KUKA KRL program: EPS_2_251806_MH46A_A_20260213065142.src

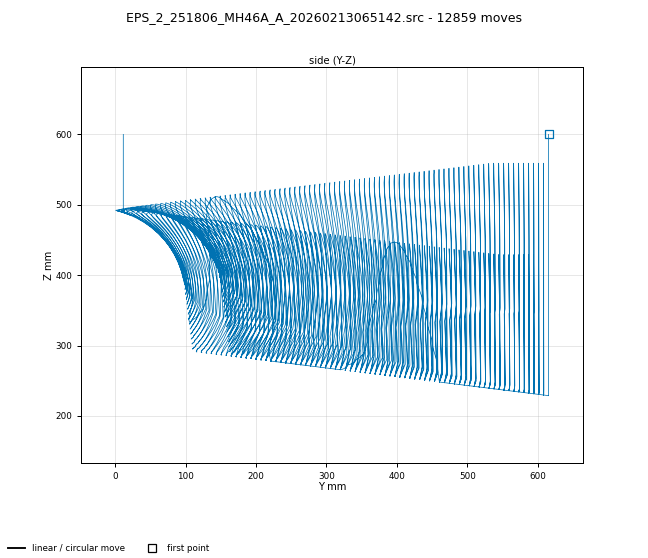
[picture p0: tool path of EPS_2_251806_MH46A_A_20260213065142.src, 12859 of 12861 moves have a stored position in this frame; points joined in program order, loops and branches not executed]
&ACCESS RVP
&REL 4
&COMMENT QRS 19112012
&PARAM EDITMASK = *
DEF PART()
EXT BAS (BAS_COMMAND :IN,REAL :IN )
INT I
BAS (#INITMOV,0 )

;KUKA QRS Post kuka4.cps  Date:22-06-2017 !

File_ID=3033

QRS_PRE_INIT()

;Init var - Until changes are made in qrs_pre_init
Outlet_Square_prg=0
Inlet_1_Square_prg=0
Inlet_2_Square_prg=0
Inlet_3_Square_prg=0
Inlet_4_Square_prg=0
Inlet_5_Square_prg=0

Outlet_1={X 0.000, Y 535.490, Z 458.500, B 0.000, E1 0.000 }
Inlet_1={X 0.000, Y 544.760, Z 328.500, B 0.000, E1 188.000 }
Outlet_1_type=201
Inlet_1_type=201
;QRS#1=Sidecore dimensions
;QRS#2=200-8" PVC SDR 35
;QRS#3=200-8" PVC SDR 35
;QRS#4=
;QRS#5=
;QRS#6=
;QRS#7=
;QRS#8=
;QRS#9=12-08 PSX
;QRS#10=12-08 PSX
;QRS#11=
;QRS#12=
;QRS#13=
;QRS#14=
;QRS#15=
;QRS#16=1220x127x838 2,75'
;QRS#17=EPS Height
;QRS#18=559
;QRS#19=*
;QRS#20= UPDATED VERSION 22-06-2017
;QRS#21=*
Outlet_Square=0100
Inlet_1_Square=0100
Inlet_2_Square=0
Inlet_3_Square=0
Inlet_4_Square=0
Inlet_5_Square=0
Mill_Square=1
Outlet_Square_Prg=204
Inlet_1_Square_prg=204

QRS_INIT()

$ADVANCE=5

; T1
PTP {E1 173.608,E2 173.608}
PTP {X 0,Y 615.502,A -85,B 0,C 180,E1 173.608,E2 173.608,E3 0,E4 0,E5 0,E6 0}
QRS_SPEED_INIT()
LIN {X 0,Y 615.502,Z 600,A -85,B 0,C 180,E1 173.608,E2 173.608,E3 0,E4 0,E5 0,E6 0} C_VEL
LIN {X 0,Y 615.502,Z 238.877,A -85,B 0,C 180,E1 173.608,E2 173.608} C_VEL
LIN {X 0,Y 615.502,Z 230.7,A -85,B 0,C 180,E1 173.608,E2 173.608} C_VEL
LIN {X 0,Y 615.471,Z 228.7,A -85,B 0,C 180,E1 173.422,E2 173.422} C_VEL
LIN {X 0,Y 615.413,Z 228.7,A -85,B 0,C 180,E1 170.8,E2 170.8} C_VEL
LIN {X 0,Y 615.412,Z 228.7,A -85,B 0,C 180,E1 168.805,E2 168.805} C_VEL
LIN {X 0,Y 615.411,Z 228.7,A -85,B 0,C 180,E1 166.797,E2 166.797} C_VEL
LIN {X 0,Y 615.451,Z 228.7,A -85,B 0,C 180,E1 164.094,E2 164.094} C_VEL
LIN {X 0,Y 615.438,Z 228.7,A -85,B 0,C 180,E1 161.352,E2 161.352} C_VEL
LIN {X 0,Y 615.424,Z 228.701,A -85,B 0,C 180,E1 159.267,E2 159.267} C_VEL
LIN {X 0,Y 615.418,Z 228.7,A -85,B 0,C 180,E1 157.152,E2 157.152} C_VEL
LIN {X 0,Y 615.412,Z 228.7,A -85,B 0,C 180,E1 155.005,E2 155.005} C_VEL
LIN {X 0,Y 615.413,Z 228.7,A -85,B 0,C 180,E1 152.819,E2 152.819} C_VEL
LIN {X 0,Y 615.467,Z 228.7,A -85,B 0,C 180,E1 150.206,E2 150.206} C_VEL
LIN {X 0,Y 615.434,Z 228.7,A -85,B 0,C 180,E1 147.539,E2 147.539} C_VEL
LIN {X 0,Y 615.411,Z 228.7,A -85,B 0,C 180,E1 145.18,E2 145.18} C_VEL
LIN {X 0,Y 615.411,Z 228.7,A -85,B 0,C 180,E1 143.071,E2 143.071} C_VEL
LIN {X 0,Y 615.415,Z 228.7,A -85,B 0,C 180,E1 140.944,E2 140.944} C_VEL
LIN {X 0,Y 615.451,Z 228.7,A -85,B 0,C 180,E1 138.523,E2 138.523} C_VEL
LIN {X 0,Y 615.443,Z 228.701,A -85,B 0,C 180,E1 135.846,E2 135.846} C_VEL
LIN {X 0,Y 615.461,Z 228.7,A -85,B 0,C 180,E1 133.994,E2 133.994} C_VEL
LIN {X 0,Y 615.414,Z 228.7,A -85,B 0,C 180,E1 131.478,E2 131.478} C_VEL
LIN {X 0,Y 615.429,Z 228.7,A -85,B 0,C 180,E1 128.907,E2 128.907} C_VEL
LIN {X 0,Y 615.472,Z 228.705,A -85,B 0,C 180,E1 126.425,E2 126.425} C_VEL
LIN {X 0,Y 615.44,Z 228.701,A -85,B 0,C 180,E1 124.024,E2 124.024} C_VEL
LIN {X 0,Y 615.416,Z 228.7,A -85,B 0,C 180,E1 121.688,E2 121.688} C_VEL
LIN {X 0,Y 615.412,Z 228.7,A -85,B 0,C 180,E1 119.409,E2 119.409} C_VEL
LIN {X 0,Y 615.435,Z 228.699,A -85,B 0,C 180,E1 117.034,E2 117.034} C_VEL
LIN {X 0,Y 615.454,Z 228.7,A -85,B 0,C 180,E1 114.273,E2 114.273} C_VEL
LIN {X 0,Y 615.436,Z 228.7,A -85,B 0,C 180,E1 112.138,E2 112.138} C_VEL
LIN {X 0,Y 615.425,Z 228.7,A -85,B 0,C 180,E1 110.034,E2 110.034} C_VEL
LIN {X 0,Y 615.418,Z 228.7,A -85,B 0,C 180,E1 107.958,E2 107.958} C_VEL
LIN {X 0,Y 615.415,Z 228.7,A -85,B 0,C 180,E1 105.906,E2 105.906} C_VEL
LIN {X 0,Y 615.413,Z 228.7,A -85,B 0,C 180,E1 103.875,E2 103.875} C_VEL
LIN {X 0,Y 615.413,Z 228.7,A -85,B 0,C 180,E1 101.862,E2 101.862} C_VEL
LIN {X 0,Y 615.412,Z 228.7,A -85,B 0,C 180,E1 99.863,E2 99.863} C_VEL
LIN {X 0,Y 615.451,Z 228.699,A -85,B 0,C 180,E1 97.216,E2 97.216} C_VEL
LIN {X 0,Y 615.493,Z 228.798,A -85,B 0,C 180,E1 94.83,E2 94.83} C_VEL
LIN {X 0,Y 615.498,Z 229.533,A -85,B 0,C 180,E1 94.707,E2 94.707} C_VEL
LIN {X 0,Y 615.499,Z 231.992,A -85,B 0,C 180,E1 94.646,E2 94.646} C_VEL
LIN {X 0,Y 615.498,Z 325.12,A -85,B 0,C 180,E1 93.539,E2 93.539} C_VEL
LIN {X 0,Y 615.497,Z 337.357,A -85,B 0,C 180,E1 93.273,E2 93.273} C_VEL
LIN {X 0,Y 615.5,Z 350.043,A -85,B 0,C 180,E1 92.863,E2 92.863} C_VEL
LIN {X 0,Y 615.492,Z 361.325,A -85,B 0,C 180,E1 92.372,E2 92.372} C_VEL
LIN {X 0,Y 615.492,Z 372.98,A -85,B 0,C 180,E1 91.717,E2 91.717} C_VEL
LIN {X 0,Y 615.498,Z 384.416,A -85,B 0,C 180,E1 90.899,E2 90.899} C_VEL
LIN {X 0,Y 615.499,Z 392.785,A -85,B 0,C 180,E1 90.163,E2 90.163} C_VEL
LIN {X 0,Y 615.497,Z 401.872,A -85,B 0,C 180,E1 89.182,E2 89.182} C_VEL
LIN {X 0,Y 615.497,Z 409.194,A -85,B 0,C 180,E1 88.2,E2 88.2} C_VEL
LIN {X 0,Y 615.497,Z 415.962,A -85,B 0,C 180,E1 87.054,E2 87.054} C_VEL
LIN {X 0,Y 615.495,Z 420.438,A -85,B 0,C 180,E1 86.071,E2 86.071} C_VEL
LIN {X 0,Y 615.497,Z 422.798,A -85,B 0,C 180,E1 85.415,E2 85.415} C_VEL
LIN {X 0,Y 615.495,Z 424.737,A -85,B 0,C 180,E1 84.759,E2 84.759} C_VEL
LIN {X 0,Y 615.499,Z 426.266,A -85,B 0,C 180,E1 84.101,E2 84.101} C_VEL
LIN {X 0,Y 615.496,Z 427.396,A -85,B 0,C 180,E1 83.42,E2 83.42} C_VEL
LIN {X 0,Y 615.497,Z 428.353,A -85,B 0,C 180,E1 82.124,E2 82.124} C_VEL
LIN {X 0,Y 615.494,Z 428.277,A -85,B 0,C 180,E1 81.463,E2 81.463} C_VEL
LIN {X 0,Y 615.497,Z 427.763,A -85,B 0,C 180,E1 80.801,E2 80.801} C_VEL
LIN {X 0,Y 615.499,Z 426.85,A -85,B 0,C 180,E1 80.138,E2 80.138} C_VEL
LIN {X 0,Y 615.494,Z 424.63,A -85,B 0,C 180,E1 79.112,E2 79.112} C_VEL
LIN {X 0,Y 615.494,Z 421.563,A -85,B 0,C 180,E1 78.139,E2 78.139} C_VEL
LIN {X 0,Y 615.498,Z 417.323,A -85,B 0,C 180,E1 77.135,E2 77.135} C_VEL
LIN {X 0,Y 615.497,Z 411.481,A -85,B 0,C 180,E1 76.066,E2 76.066} C_VEL
LIN {X 0,Y 615.496,Z 404.939,A -85,B 0,C 180,E1 75.113,E2 75.113} C_VEL
LIN {X 0,Y 615.499,Z 397.838,A -85,B 0,C 180,E1 74.265,E2 74.265} C_VEL
LIN {X 0,Y 615.497,Z 389.203,A -85,B 0,C 180,E1 73.414,E2 73.414} C_VEL
LIN {X 0,Y 615.497,Z 378.418,A -85,B 0,C 180,E1 72.559,E2 72.559} C_VEL
LIN {X 0,Y 615.484,Z 367.8,A -85,B 0,C 180,E1 71.881,E2 71.881} C_VEL
LIN {X 0,Y 615.498,Z 357.473,A -85,B 0,C 180,E1 71.354,E2 71.354} C_VEL
LIN {X 0,Y 615.498,Z 345.389,A -85,B 0,C 180,E1 70.879,E2 70.879} C_VEL
LIN {X 0,Y 615.499,Z 333.141,A -85,B 0,C 180,E1 70.533,E2 70.533} C_VEL
LIN {X 0,Y 615.497,Z 319.785,A -85,B 0,C 180,E1 70.294,E2 70.294} C_VEL
LIN {X 0,Y 615.499,Z 229.907,A -85,B 0,C 180,E1 69.226,E2 69.226} C_VEL
LIN {X 0,Y 615.499,Z 228.833,A -85,B 0,C 180,E1 69.095,E2 69.095} C_VEL
LIN {X 0,Y 615.442,Z 228.696,A -85,B 0,C 180,E1 66.442,E2 66.442} C_VEL
LIN {X 0,Y 615.437,Z 228.695,A -85,B 0,C 180,E1 64.282,E2 64.282} C_VEL
LIN {X 0,Y 615.487,Z 228.69,A -85,B 0,C 180,E1 61.551,E2 61.551} C_VEL
LIN {X 0,Y 615.464,Z 228.698,A -85,B 0,C 180,E1 58.919,E2 58.919} C_VEL
LIN {X 0,Y 615.435,Z 228.695,A -85,B 0,C 180,E1 56.474,E2 56.474} C_VEL
LIN {X 0,Y 615.442,Z 228.693,A -85,B 0,C 180,E1 54.173,E2 54.173} C_VEL
LIN {X 0,Y 615.463,Z 228.692,A -85,B 0,C 180,E1 51.93,E2 51.93} C_VEL
LIN {X 0,Y 615.487,Z 228.703,A -85,B 0,C 180,E1 49.394,E2 49.394} C_VEL
LIN {X 0,Y 615.436,Z 228.696,A -85,B 0,C 180,E1 46.752,E2 46.752} C_VEL
LIN {X 0,Y 615.468,Z 228.692,A -85,B 0,C 180,E1 43.997,E2 43.997} C_VEL
LIN {X 0,Y 615.448,Z 228.698,A -85,B 0,C 180,E1 41.091,E2 41.091} C_VEL
LIN {X 0,Y 615.434,Z 228.697,A -85,B 0,C 180,E1 38.909,E2 38.909} C_VEL
LIN {X 0,Y 615.442,Z 228.694,A -85,B 0,C 180,E1 36.428,E2 36.428} C_VEL
LIN {X 0,Y 615.481,Z 228.693,A -85,B 0,C 180,E1 34.023,E2 34.023} C_VEL
LIN {X 0,Y 615.435,Z 228.697,A -85,B 0,C 180,E1 31.079,E2 31.079} C_VEL
LIN {X 0,Y 615.436,Z 228.695,A -85,B 0,C 180,E1 28.661,E2 28.661} C_VEL
LIN {X 0,Y 615.482,Z 228.699,A -85,B 0,C 180,E1 25.716,E2 25.716} C_VEL
LIN {X 0,Y 615.458,Z 228.699,A -85,B 0,C 180,E1 23.558,E2 23.558} C_VEL
LIN {X 0,Y 615.443,Z 228.698,A -85,B 0,C 180,E1 21.434,E2 21.434} C_VEL
LIN {X 0,Y 615.435,Z 228.697,A -85,B 0,C 180,E1 19.34,E2 19.34} C_VEL
LIN {X 0,Y 615.43,Z 228.697,A -85,B 0,C 180,E1 17.272,E2 17.272} C_VEL
LIN {X 0,Y 615.428,Z 228.697,A -85,B 0,C 180,E1 15.228,E2 15.228} C_VEL
LIN {X 0,Y 615.427,Z 228.697,A -85,B 0,C 180,E1 13.203,E2 13.203} C_VEL
LIN {X 0,Y 615.471,Z 228.694,A -85,B 0,C 180,E1 10.527,E2 10.527} C_VEL
LIN {X 0,Y 615.459,Z 228.699,A -85,B 0,C 180,E1 7.876,E2 7.876} C_VEL
LIN {X 0,Y 615.426,Z 228.696,A -85,B 0,C 180,E1 5.242,E2 5.242} C_VEL
LIN {X 0,Y 615.476,Z 228.694,A -85,B 0,C 180,E1 2.618,E2 2.618} C_VEL
LIN {X 0,Y 615.455,Z 228.699,A -85,B 0,C 180,E1 0,E2 0} C_VEL
LIN {X 0,Y 615.422,Z 228.697,A -85,B 0,C 180,E1 -2.618,E2 -2.618} C_VEL
LIN {X 0,Y 615.475,Z 228.695,A -85,B 0,C 180,E1 -5.241,E2 -5.241} C_VEL
LIN {X 0,Y 615.452,Z 228.699,A -85,B 0,C 180,E1 -7.876,E2 -7.876} C_VEL
LIN {X 0,Y 615.449,Z 228.699,A -85,B 0,C 180,E1 -9.863,E2 -9.863} C_VEL
LIN {X 0,Y 615.446,Z 228.699,A -85,B 0,C 180,E1 -11.862,E2 -11.862} C_VEL
LIN {X 0,Y 615.437,Z 228.699,A -85,B 0,C 180,E1 -13.918,E2 -13.918} C_VEL
LIN {X 0,Y 615.435,Z 228.699,A -85,B 0,C 180,E1 -15.907,E2 -15.907} C_VEL
LIN {X 0,Y 615.428,Z 228.699,A -85,B 0,C 180,E1 -17.959,E2 -17.959} C_VEL
LIN {X 0,Y 615.424,Z 228.698,A -85,B 0,C 180,E1 -20.035,E2 -20.035} C_VEL
LIN {X 0,Y 615.422,Z 228.698,A -85,B 0,C 180,E1 -22.334,E2 -22.334} C_VEL
LIN {X 0,Y 615.486,Z 228.696,A -85,B 0,C 180,E1 -24.992,E2 -24.992} C_VEL
LIN {X 0,Y 615.485,Z 228.702,A -85,B 0,C 180,E1 -27.177,E2 -27.177} C_VEL
LIN {X 0,Y 615.425,Z 228.699,A -85,B 0,C 180,E1 -29.786,E2 -29.786} C_VEL
LIN {X 0,Y 615.427,Z 228.699,A -85,B 0,C 180,E1 -31.689,E2 -31.689} C_VEL
LIN {X 0,Y 615.418,Z 228.698,A -85,B 0,C 180,E1 -34.026,E2 -34.026} C_VEL
LIN {X 0,Y 615.439,Z 228.698,A -85,B 0,C 180,E1 -36.428,E2 -36.428} C_VEL
LIN {X 0,Y 615.477,Z 228.7,A -85,B 0,C 180,E1 -39.062,E2 -39.062} C_VEL
LIN {X 0,Y 615.427,Z 228.699,A -85,B 0,C 180,E1 -41.479,E2 -41.479} C_VEL
LIN {X 0,Y 615.419,Z 228.699,A -85,B 0,C 180,E1 -43.992,E2 -43.992} C_VEL
LIN {X 0,Y 615.499,Z 228.7,A -85,B 0,C 180,E1 -46.757,E2 -46.757} C_VEL
LIN {X 0,Y 615.422,Z 228.7,A -85,B 0,C 180,E1 -49.389,E2 -49.389} C_VEL
LIN {X 0,Y 615.424,Z 228.699,A -85,B 0,C 180,E1 -51.996,E2 -51.996} C_VEL
LIN {X 0,Y 615.467,Z 228.699,A -85,B 0,C 180,E1 -54.383,E2 -54.383} C_VEL
LIN {X 0,Y 615.471,Z 228.7,A -85,B 0,C 180,E1 -56.763,E2 -56.763} C_VEL
LIN {X 0,Y 615.43,Z 228.7,A -85,B 0,C 180,E1 -59.078,E2 -59.078} C_VEL
LIN {X 0,Y 615.414,Z 228.7,A -85,B 0,C 180,E1 -61.339,E2 -61.339} C_VEL
LIN {X 0,Y 615.41,Z 228.7,A -85,B 0,C 180,E1 -63.553,E2 -63.553} C_VEL
LIN {X 0,Y 615.499,Z 228.856,A -85,B 0,C 180,E1 -64.539,E2 -64.539} C_VEL
LIN {X 0,Y 615.497,Z 231.379,A -85,B 0,C 180,E1 -64.864,E2 -64.864} C_VEL
LIN {X 0,Y 615.489,Z 256.529,A -85,B 0,C 180,E1 -67.654,E2 -67.654} C_VEL
LIN {X 0,Y 615.496,Z 282.599,A -85,B 0,C 180,E1 -70.489,E2 -70.489} C_VEL
LIN {X 0,Y 615.493,Z 309.957,A -85,B 0,C 180,E1 -73.414,E2 -73.414} C_VEL
LIN {X 0,Y 615.487,Z 337.276,A -85,B 0,C 180,E1 -76.294,E2 -76.294} C_VEL
LIN {X 0,Y 615.498,Z 345.12,A -85,B 0,C 180,E1 -77.093,E2 -77.093} C_VEL
LIN {X 0,Y 615.491,Z 454.828,A -85,B 0,C 180,E1 -78.411,E2 -78.411} C_VEL
LIN {X 0,Y 615.499,Z 467.341,A -85,B 0,C 180,E1 -78.682,E2 -78.682} C_VEL
LIN {X 0,Y 615.496,Z 480.499,A -85,B 0,C 180,E1 -79.109,E2 -79.109} C_VEL
LIN {X 0,Y 615.48,Z 492.477,A -85,B 0,C 180,E1 -79.639,E2 -79.639} C_VEL
LIN {X 0,Y 615.493,Z 503.993,A -85,B 0,C 180,E1 -80.304,E2 -80.304} C_VEL
LIN {X 0,Y 615.499,Z 514.34,A -85,B 0,C 180,E1 -81.05,E2 -81.05} C_VEL
LIN {X 0,Y 615.497,Z 522.811,A -85,B 0,C 180,E1 -81.794,E2 -81.794} C_VEL
LIN {X 0,Y 615.498,Z 530.605,A -85,B 0,C 180,E1 -82.619,E2 -82.619} C_VEL
LIN {X 0,Y 615.496,Z 538.202,A -85,B 0,C 180,E1 -83.608,E2 -83.608} C_VEL
LIN {X 0,Y 615.498,Z 545.204,A -85,B 0,C 180,E1 -84.759,E2 -84.759} C_VEL
LIN {X 0,Y 615.493,Z 549.851,A -85,B 0,C 180,E1 -85.743,E2 -85.743} C_VEL
LIN {X 0,Y 615.495,Z 553.398,A -85,B 0,C 180,E1 -86.727,E2 -86.727} C_VEL
LIN {X 0,Y 615.497,Z 555.232,A -85,B 0,C 180,E1 -87.382,E2 -87.382} C_VEL
LIN {X 0,Y 615.499,Z 556.607,A -85,B 0,C 180,E1 -88.037,E2 -88.037} C_VEL
LIN {X 0,Y 615.496,Z 558.173,A -85,B 0,C 180,E1 -89.345,E2 -89.345} C_VEL
LIN {X 0,Y 615.494,Z 558.389,A -85,B 0,C 180,E1 -90,E2 -90} C_VEL
LIN {X 0,Y 615.496,Z 557.58,A -85,B 0,C 180,E1 -91.308,E2 -91.308} C_VEL
LIN {X 0,Y 615.499,Z 556.608,A -85,B 0,C 180,E1 -91.963,E2 -91.963} C_VEL
LIN {X 0,Y 615.497,Z 555.234,A -85,B 0,C 180,E1 -92.617,E2 -92.617} C_VEL
LIN {X 0,Y 615.496,Z 552.351,A -85,B 0,C 180,E1 -93.6,E2 -93.6} C_VEL
LIN {X 0,Y 615.498,Z 548.443,A -85,B 0,C 180,E1 -94.584,E2 -94.584} C_VEL
LIN {X 0,Y 615.499,Z 543.407,A -85,B 0,C 180,E1 -95.569,E2 -95.569} C_VEL
LIN {X 0,Y 615.496,Z 536.869,A -85,B 0,C 180,E1 -96.583,E2 -96.583} C_VEL
LIN {X 0,Y 615.497,Z 529.137,A -85,B 0,C 180,E1 -97.545,E2 -97.545} C_VEL
LIN {X 0,Y 615.498,Z 521.05,A -85,B 0,C 180,E1 -98.371,E2 -98.371} C_VEL
LIN {X 0,Y 615.499,Z 511.174,A -85,B 0,C 180,E1 -99.198,E2 -99.198} C_VEL
LIN {X 0,Y 615.492,Z 499.989,A -85,B 0,C 180,E1 -99.945,E2 -99.945} C_VEL
LIN {X 0,Y 615.485,Z 489.034,A -85,B 0,C 180,E1 -100.526,E2 -100.526} C_VEL
LIN {X 0,Y 615.499,Z 476.423,A -85,B 0,C 180,E1 -101.042,E2 -101.042} C_VEL
LIN {X 0,Y 615.498,Z 464.086,A -85,B 0,C 180,E1 -101.401,E2 -101.401} C_VEL
LIN {X 0,Y 615.491,Z 450.504,A -85,B 0,C 180,E1 -101.651,E2 -101.651} C_VEL
LIN {X 0,Y 615.498,Z 345.13,A -85,B 0,C 180,E1 -102.907,E2 -102.907} C_VEL
LIN {X 0,Y 615.487,Z 319.609,A -85,B 0,C 180,E1 -105.565,E2 -105.565} C_VEL
LIN {X 0,Y 615.483,Z 292.55,A -85,B 0,C 180,E1 -108.442,E2 -108.442} C_VEL
LIN {X 0,Y 615.483,Z 266.498,A -85,B 0,C 180,E1 -111.256,E2 -111.256} C_VEL
LIN {X 0,Y 615.498,Z 240.288,A -85,B 0,C 180,E1 -114.14,E2 -114.14} C_VEL
LIN {X 0,Y 615.499,Z 228.979,A -85,B 0,C 180,E1 -115.425,E2 -115.425} C_VEL
LIN {X 0,Y 615.473,Z 228.701,A -85,B 0,C 180,E1 -115.715,E2 -115.715} C_VEL
LIN {X 0,Y 615.411,Z 228.7,A -85,B 0,C 180,E1 -118.437,E2 -118.437} C_VEL
LIN {X 0,Y 615.421,Z 228.7,A -85,B 0,C 180,E1 -120.163,E2 -120.163} C_VEL
LIN {X 0,Y 615.411,Z 228.7,A -85,B 0,C 180,E1 -122.461,E2 -122.461} C_VEL
LIN {X 0,Y 615.425,Z 228.7,A -85,B 0,C 180,E1 -124.818,E2 -124.818} C_VEL
LIN {X 0,Y 615.471,Z 228.702,A -85,B 0,C 180,E1 -127.242,E2 -127.242} C_VEL
LIN {X 0,Y 615.414,Z 228.7,A -85,B 0,C 180,E1 -130.081,E2 -130.081} C_VEL
LIN {X 0,Y 615.41,Z 228.7,A -85,B 0,C 180,E1 -132.358,E2 -132.358} C_VEL
LIN {X 0,Y 615.411,Z 228.7,A -85,B 0,C 180,E1 -134.155,E2 -134.155} C_VEL
LIN {X 0,Y 615.436,Z 228.7,A -85,B 0,C 180,E1 -136.751,E2 -136.751} C_VEL
LIN {X 0,Y 615.459,Z 228.702,A -85,B 0,C 180,E1 -139.391,E2 -139.391} C_VEL
LIN {X 0,Y 615.412,Z 228.7,A -85,B 0,C 180,E1 -141.995,E2 -141.995} C_VEL
LIN {X 0,Y 615.418,Z 228.7,A -85,B 0,C 180,E1 -144.379,E2 -144.379} C_VEL
LIN {X 0,Y 615.456,Z 228.7,A -85,B 0,C 180,E1 -146.762,E2 -146.762} C_VEL
LIN {X 0,Y 615.475,Z 228.703,A -85,B 0,C 180,E1 -149.08,E2 -149.08} C_VEL
LIN {X 0,Y 615.426,Z 228.7,A -85,B 0,C 180,E1 -151.557,E2 -151.557} C_VEL
LIN {X 0,Y 615.424,Z 228.7,A -85,B 0,C 180,E1 -153.553,E2 -153.553} C_VEL
LIN {X 0,Y 615.413,Z 228.7,A -85,B 0,C 180,E1 -155.725,E2 -155.725} C_VEL
LIN {X 0,Y 615.41,Z 228.7,A -85,B 0,C 180,E1 -157.861,E2 -157.861} C_VEL
LIN {X 0,Y 615.474,Z 228.7,A -85,B 0,C 180,E1 -160.662,E2 -160.662} C_VEL
LIN {X 0,Y 615.422,Z 228.7,A -85,B 0,C 180,E1 -163.412,E2 -163.412} C_VEL
LIN {X 0,Y 615.418,Z 228.7,A -85,B 0,C 180,E1 -165.449,E2 -165.449} C_VEL
LIN {X 0,Y 615.416,Z 228.7,A -85,B 0,C 180,E1 -167.468,E2 -167.468} C_VEL
LIN {X 0,Y 615.414,Z 228.7,A -85,B 0,C 180,E1 -169.472,E2 -169.472} C_VEL
LIN {X 0,Y 615.413,Z 228.7,A -85,B 0,C 180,E1 -171.462,E2 -171.462} C_VEL
LIN {X 0,Y 615.412,Z 228.7,A -85,B 0,C 180,E1 -173.469,E2 -173.469} C_VEL
LIN {X 0,Y 615.413,Z 228.7,A -85,B 0,C 180,E1 -175.415,E2 -175.415} C_VEL
LIN {X 0,Y 615.413,Z 228.7,A -85,B 0,C 180,E1 -177.382,E2 -177.382} C_VEL
LIN {X 0,Y 615.413,Z 228.7,A -85,B 0,C 180,E1 -179.346,E2 -179.346} C_VEL
LIN {X 0,Y 615.413,Z 228.7,A -85,B 0,C 180,E1 -181.309,E2 -181.309} C_VEL
LIN {X 0,Y 615.414,Z 228.7,A -85,B 0,C 180,E1 -183.274,E2 -183.274} C_VEL
LIN {X 0,Y 615.414,Z 228.7,A -85,B 0,C 180,E1 -185.242,E2 -185.242} C_VEL
LIN {X 0,Y 615.471,Z 228.7,A -85,B 0,C 180,E1 -186.578,E2 -186.578} C_VEL
LIN {X 0,Y 614.756,Z 228.843,A -85,B 0,C 180,E1 -187.124,E2 -187.124} C_VEL
LIN {X 0,Y 611.893,Z 229.263,A -85,B 0,C 180,E1 -188.01,E2 -188.01} C_VEL
LIN {X 0,Y 609.505,Z 229.569,A -85,B 0,C 180,E1 -188.722,E2 -188.722} C_VEL
LIN {X 0,Y 608.483,Z 229.685,A -85,B 0,C 180,E1 -189.272,E2 -189.272} C_VEL
LIN {X 0,Y 608.399,Z 229.694,A -85,B 0,C 180,E1 -189.458,E2 -189.458} C_VEL
LIN {X 0,Y 608.422,Z 229.696,A -85,B 0,C 180,E1 -192.001,E2 -192.001} C_VEL
LIN {X 0,Y 608.408,Z 229.696,A -85,B 0,C 180,E1 -194.722,E2 -194.722} C_VEL
LIN {X 0,Y 608.406,Z 229.695,A -85,B 0,C 180,E1 -196.786,E2 -196.786} C_VEL
LIN {X 0,Y 608.406,Z 229.695,A -85,B 0,C 180,E1 -199.572,E2 -199.572} C_VEL
LIN {X 0,Y 608.431,Z 229.695,A -85,B 0,C 180,E1 -202.474,E2 -202.474} C_VEL
LIN {X 0,Y 608.418,Z 229.695,A -85,B 0,C 180,E1 -204.573,E2 -204.573} C_VEL
LIN {X 0,Y 608.396,Z 229.695,A -85,B 0,C 180,E1 -207.195,E2 -207.195} C_VEL
LIN {X 0,Y 608.452,Z 229.698,A -85,B 0,C 180,E1 -209.972,E2 -209.972} C_VEL
LIN {X 0,Y 608.405,Z 229.693,A -85,B 0,C 180,E1 -212.883,E2 -212.883} C_VEL
LIN {X 0,Y 608.399,Z 229.695,A -85,B 0,C 180,E1 -215.281,E2 -215.281} C_VEL
LIN {X 0,Y 608.413,Z 229.697,A -85,B 0,C 180,E1 -218.236,E2 -218.236} C_VEL
LIN {X 0,Y 608.425,Z 229.694,A -85,B 0,C 180,E1 -220.328,E2 -220.328} C_VEL
LIN {X 0,Y 608.386,Z 229.696,A -85,B 0,C 180,E1 -222.966,E2 -222.966} C_VEL
LIN {X 0,Y 608.446,Z 229.699,A -85,B 0,C 180,E1 -225.738,E2 -225.738} C_VEL
LIN {X 0,Y 608.449,Z 229.695,A -85,B 0,C 180,E1 -227.939,E2 -227.939} C_VEL
LIN {X 0,Y 608.395,Z 229.695,A -85,B 0,C 180,E1 -230.712,E2 -230.712} C_VEL
LIN {X 0,Y 608.401,Z 229.696,A -85,B 0,C 180,E1 -233.083,E2 -233.083} C_VEL
LIN {X 0,Y 608.439,Z 229.699,A -85,B 0,C 180,E1 -235.53,E2 -235.53} C_VEL
LIN {X 0,Y 608.442,Z 229.693,A -85,B 0,C 180,E1 -237.905,E2 -237.905} C_VEL
LIN {X 0,Y 608.408,Z 229.694,A -85,B 0,C 180,E1 -240.218,E2 -240.218} C_VEL
LIN {X 0,Y 608.4,Z 229.694,A -85,B 0,C 180,E1 -242.481,E2 -242.481} C_VEL
LIN {X 0,Y 608.422,Z 229.702,A -85,B 0,C 180,E1 -245.429,E2 -245.429} C_VEL
LIN {X 0,Y 608.386,Z 229.696,A -85,B 0,C 180,E1 -248.306,E2 -248.306} C_VEL
LIN {X 0,Y 608.395,Z 229.695,A -85,B 0,C 180,E1 -250.428,E2 -250.428} C_VEL
LIN {X 0,Y 608.432,Z 229.699,A -85,B 0,C 180,E1 -253.216,E2 -253.216} C_VEL
LIN {X 0,Y 608.403,Z 229.694,A -85,B 0,C 180,E1 -256.01,E2 -256.01} C_VEL
LIN {X 0,Y 608.408,Z 229.694,A -85,B 0,C 180,E1 -258,E2 -258} C_VEL
LIN {X 0,Y 608.395,Z 229.695,A -85,B 0,C 180,E1 -260.022,E2 -260.022} C_VEL
LIN {X 0,Y 608.42,Z 229.695,A -85,B 0,C 180,E1 -262.701,E2 -262.701} C_VEL
LIN {X 0,Y 608.495,Z 229.908,A -85,B 0,C 180,E1 -265.093,E2 -265.093} C_VEL
LIN {X 0,Y 608.613,Z 230.708,A -85,B 0,C 180,E1 -265.177,E2 -265.177} C_VEL
LIN {X 0,Y 608.558,Z 325.816,A -85,B 0,C 180,E1 -266.338,E2 -266.338} C_VEL
LIN {X 0,Y 608.533,Z 339.357,A -85,B 0,C 180,E1 -266.649,E2 -266.649} C_VEL
LIN {X 0,Y 608.54,Z 351.561,A -85,B 0,C 180,E1 -267.063,E2 -267.063} C_VEL
LIN {X 0,Y 608.512,Z 363.321,A -85,B 0,C 180,E1 -267.601,E2 -267.601} C_VEL
LIN {X 0,Y 608.488,Z 374.605,A -85,B 0,C 180,E1 -268.263,E2 -268.263} C_VEL
LIN {X 0,Y 608.477,Z 384.808,A -85,B 0,C 180,E1 -269.008,E2 -269.008} C_VEL
LIN {X 0,Y 608.469,Z 394.048,A -85,B 0,C 180,E1 -269.835,E2 -269.835} C_VEL
LIN {X 0,Y 608.473,Z 402.998,A -85,B 0,C 180,E1 -270.828,E2 -270.828} C_VEL
LIN {X 0,Y 608.445,Z 410.246,A -85,B 0,C 180,E1 -271.821,E2 -271.821} C_VEL
LIN {X 0,Y 608.451,Z 416.901,A -85,B 0,C 180,E1 -272.98,E2 -272.98} C_VEL
LIN {X 0,Y 608.433,Z 421.316,A -85,B 0,C 180,E1 -273.974,E2 -273.974} C_VEL
LIN {X 0,Y 608.429,Z 423.649,A -85,B 0,C 180,E1 -274.638,E2 -274.638} C_VEL
LIN {X 0,Y 608.438,Z 425.558,A -85,B 0,C 180,E1 -275.302,E2 -275.302} C_VEL
LIN {X 0,Y 608.435,Z 427.045,A -85,B 0,C 180,E1 -275.967,E2 -275.967} C_VEL
LIN {X 0,Y 608.43,Z 428.08,A -85,B 0,C 180,E1 -276.633,E2 -276.633} C_VEL
LIN {X 0,Y 608.422,Z 428.988,A -85,B 0,C 180,E1 -277.968,E2 -277.968} C_VEL
LIN {X 0,Y 608.418,Z 428.833,A -85,B 0,C 180,E1 -278.637,E2 -278.637} C_VEL
LIN {X 0,Y 608.434,Z 427.29,A -85,B 0,C 180,E1 -279.978,E2 -279.978} C_VEL
LIN {X 0,Y 608.423,Z 425.177,A -85,B 0,C 180,E1 -280.931,E2 -280.931} C_VEL
LIN {X 0,Y 608.444,Z 421.747,A -85,B 0,C 180,E1 -282,E2 -282} C_VEL
LIN {X 0,Y 608.431,Z 417.354,A -85,B 0,C 180,E1 -283.017,E2 -283.017} C_VEL
LIN {X 0,Y 608.437,Z 411.708,A -85,B 0,C 180,E1 -284.038,E2 -284.038} C_VEL
LIN {X 0,Y 608.446,Z 404.606,A -85,B 0,C 180,E1 -285.064,E2 -285.064} C_VEL
LIN {X 0,Y 608.462,Z 395.62,A -85,B 0,C 180,E1 -286.094,E2 -286.094} C_VEL
LIN {X 0,Y 608.485,Z 386.349,A -85,B 0,C 180,E1 -286.956,E2 -286.956} C_VEL
LIN {X 0,Y 608.49,Z 375.995,A -85,B 0,C 180,E1 -287.736,E2 -287.736} C_VEL
LIN {X 0,Y 608.495,Z 364.675,A -85,B 0,C 180,E1 -288.417,E2 -288.417} C_VEL
LIN {X 0,Y 608.519,Z 352.285,A -85,B 0,C 180,E1 -288.999,E2 -288.999} C_VEL
LIN {X 0,Y 608.543,Z 339.557,A -85,B 0,C 180,E1 -289.436,E2 -289.436} C_VEL
LIN {X 0,Y 608.553,Z 326.329,A -85,B 0,C 180,E1 -289.743,E2 -289.743} C_VEL
LIN {X 0,Y 608.57,Z 293.063,A -85,B 0,C 180,E1 -290.16,E2 -290.16} C_VEL
LIN {X 0,Y 608.597,Z 230.787,A -85,B 0,C 180,E1 -290.909,E2 -290.909} C_VEL
LIN {X 0,Y 608.495,Z 229.799,A -85,B 0,C 180,E1 -291.024,E2 -291.024} C_VEL
LIN {X 0,Y 608.426,Z 229.691,A -85,B 0,C 180,E1 -293.846,E2 -293.846} C_VEL
LIN {X 0,Y 608.442,Z 229.698,A -85,B 0,C 180,E1 -296.774,E2 -296.774} C_VEL
LIN {X 0,Y 608.426,Z 229.698,A -85,B 0,C 180,E1 -299.022,E2 -299.022} C_VEL
LIN {X 0,Y 608.434,Z 229.692,A -85,B 0,C 180,E1 -301.318,E2 -301.318} C_VEL
LIN {X 0,Y 608.425,Z 229.691,A -85,B 0,C 180,E1 -303.727,E2 -303.727} C_VEL
LIN {X 0,Y 608.438,Z 229.691,A -85,B 0,C 180,E1 -306.092,E2 -306.092} C_VEL
LIN {X 0,Y 608.42,Z 229.701,A -85,B 0,C 180,E1 -308.591,E2 -308.591} C_VEL
LIN {X 0,Y 608.419,Z 229.692,A -85,B 0,C 180,E1 -311.337,E2 -311.337} C_VEL
LIN {X 0,Y 608.448,Z 229.689,A -85,B 0,C 180,E1 -313.87,E2 -313.87} C_VEL
LIN {X 0,Y 608.456,Z 229.694,A -85,B 0,C 180,E1 -316.692,E2 -316.692} C_VEL
LIN {X 0,Y 608.429,Z 229.691,A -85,B 0,C 180,E1 -319.672,E2 -319.672} C_VEL
LIN {X 0,Y 608.453,Z 229.696,A -85,B 0,C 180,E1 -322.252,E2 -322.252} C_VEL
LIN {X 0,Y 608.428,Z 229.695,A -85,B 0,C 180,E1 -324.721,E2 -324.721} C_VEL
LIN {X 0,Y 608.421,Z 229.692,A -85,B 0,C 180,E1 -327.118,E2 -327.118} C_VEL
LIN {X 0,Y 608.471,Z 229.692,A -85,B 0,C 180,E1 -330.026,E2 -330.026} C_VEL
LIN {X 0,Y 608.414,Z 229.694,A -85,B 0,C 180,E1 -332.803,E2 -332.803} C_VEL
LIN {X 0,Y 608.426,Z 229.692,A -85,B 0,C 180,E1 -335.427,E2 -335.427} C_VEL
LIN {X 0,Y 608.446,Z 229.694,A -85,B 0,C 180,E1 -338.307,E2 -338.307} C_VEL
LIN {X 0,Y 608.426,Z 229.691,A -85,B 0,C 180,E1 -341.129,E2 -341.129} C_VEL
LIN {X 0,Y 608.452,Z 229.697,A -85,B 0,C 180,E1 -343.906,E2 -343.906} C_VEL
LIN {X 0,Y 608.418,Z 229.693,A -85,B 0,C 180,E1 -346.642,E2 -346.642} C_VEL
LIN {X 0,Y 608.438,Z 229.692,A -85,B 0,C 180,E1 -349.349,E2 -349.349} C_VEL
LIN {X 0,Y 608.454,Z 229.694,A -85,B 0,C 180,E1 -352.033,E2 -352.033} C_VEL
LIN {X 0,Y 608.411,Z 229.693,A -85,B 0,C 180,E1 -354.697,E2 -354.697} C_VEL
LIN {X 0,Y 608.465,Z 229.69,A -85,B 0,C 180,E1 -357.352,E2 -357.352} C_VEL
LIN {X 0,Y 608.448,Z 229.693,A -85,B 0,C 180,E1 -360,E2 -360} C_VEL
LIN {X 0,Y 608.42,Z 229.691,A -85,B 0,C 180,E1 -362.648,E2 -362.648} C_VEL
LIN {X 0,Y 608.452,Z 229.693,A -85,B 0,C 180,E1 -365.302,E2 -365.302} C_VEL
LIN {X 0,Y 608.414,Z 229.695,A -85,B 0,C 180,E1 -367.968,E2 -367.968} C_VEL
LIN {X 0,Y 608.417,Z 229.695,A -85,B 0,C 180,E1 -369.978,E2 -369.978} C_VEL
LIN {X 0,Y 608.421,Z 229.693,A -85,B 0,C 180,E1 -372.001,E2 -372.001} C_VEL
LIN {X 0,Y 608.409,Z 229.694,A -85,B 0,C 180,E1 -374.039,E2 -374.039} C_VEL
LIN {X 0,Y 608.397,Z 229.695,A -85,B 0,C 180,E1 -376.51,E2 -376.51} C_VEL
LIN {X 0,Y 608.43,Z 229.694,A -85,B 0,C 180,E1 -378.87,E2 -378.87} C_VEL
LIN {X 0,Y 608.437,Z 229.693,A -85,B 0,C 180,E1 -381.693,E2 -381.693} C_VEL
LIN {X 0,Y 608.421,Z 229.693,A -85,B 0,C 180,E1 -384.572,E2 -384.572} C_VEL
LIN {X 0,Y 608.458,Z 229.696,A -85,B 0,C 180,E1 -387.205,E2 -387.205} C_VEL
LIN {X 0,Y 608.393,Z 229.695,A -85,B 0,C 180,E1 -389.961,E2 -389.961} C_VEL
LIN {X 0,Y 608.418,Z 229.694,A -85,B 0,C 180,E1 -392.517,E2 -392.517} C_VEL
LIN {X 0,Y 608.409,Z 229.698,A -85,B 0,C 180,E1 -395.28,E2 -395.28} C_VEL
LIN {X 0,Y 608.397,Z 229.695,A -85,B 0,C 180,E1 -397.752,E2 -397.752} C_VEL
LIN {X 0,Y 608.427,Z 229.693,A -85,B 0,C 180,E1 -400.327,E2 -400.327} C_VEL
LIN {X 0,Y 608.435,Z 229.693,A -85,B 0,C 180,E1 -403.306,E2 -403.306} C_VEL
LIN {X 0,Y 608.42,Z 229.693,A -85,B 0,C 180,E1 -406.127,E2 -406.127} C_VEL
LIN {X 0,Y 608.439,Z 229.698,A -85,B 0,C 180,E1 -408.823,E2 -408.823} C_VEL
LIN {X 0,Y 608.393,Z 229.696,A -85,B 0,C 180,E1 -411.407,E2 -411.407} C_VEL
LIN {X 0,Y 608.403,Z 229.694,A -85,B 0,C 180,E1 -413.905,E2 -413.905} C_VEL
LIN {X 0,Y 608.441,Z 229.695,A -85,B 0,C 180,E1 -416.328,E2 -416.328} C_VEL
LIN {X 0,Y 608.432,Z 229.697,A -85,B 0,C 180,E1 -418.735,E2 -418.735} C_VEL
LIN {X 0,Y 608.383,Z 229.696,A -85,B 0,C 180,E1 -421.396,E2 -421.396} C_VEL
LIN {X 0,Y 608.409,Z 229.698,A -85,B 0,C 180,E1 -423.963,E2 -423.963} C_VEL
LIN {X 0,Y 608.513,Z 229.951,A -85,B 0,C 180,E1 -424.383,E2 -424.383} C_VEL
LIN {X 0,Y 608.694,Z 237.5,A -85,B 0,C 180,E1 -425.258,E2 -425.258} C_VEL
LIN {X 0,Y 608.634,Z 263.271,A -85,B 0,C 180,E1 -428.137,E2 -428.137} C_VEL
LIN {X 0,Y 608.577,Z 289.043,A -85,B 0,C 180,E1 -430.96,E2 -430.96} C_VEL
LIN {X 0,Y 608.549,Z 315.181,A -85,B 0,C 180,E1 -433.776,E2 -433.776} C_VEL
LIN {X 0,Y 608.483,Z 340.585,A -85,B 0,C 180,E1 -436.474,E2 -436.474} C_VEL
LIN {X 0,Y 608.533,Z 345.16,A -85,B 0,C 180,E1 -436.943,E2 -436.943} C_VEL
LIN {X 0,Y 608.583,Z 363.241,A -85,B 0,C 180,E1 -437.177,E2 -437.177} C_VEL
LIN {X 0,Y 608.542,Z 454.946,A -85,B 0,C 180,E1 -438.277,E2 -438.277} C_VEL
LIN {X 0,Y 608.546,Z 468.215,A -85,B 0,C 180,E1 -438.572,E2 -438.572} C_VEL
LIN {X 0,Y 608.544,Z 481.33,A -85,B 0,C 180,E1 -439.009,E2 -439.009} C_VEL
LIN {X 0,Y 608.502,Z 492.634,A -85,B 0,C 180,E1 -439.519,E2 -439.519} C_VEL
LIN {X 0,Y 608.487,Z 504.196,A -85,B 0,C 180,E1 -440.191,E2 -440.191} C_VEL
LIN {X 0,Y 608.485,Z 514.593,A -85,B 0,C 180,E1 -440.946,E2 -440.946} C_VEL
LIN {X 0,Y 608.475,Z 523.111,A -85,B 0,C 180,E1 -441.699,E2 -441.699} C_VEL
LIN {X 0,Y 608.471,Z 530.959,A -85,B 0,C 180,E1 -442.534,E2 -442.534} C_VEL
LIN {X 0,Y 608.461,Z 538.286,A -85,B 0,C 180,E1 -443.484,E2 -443.484} C_VEL
LIN {X 0,Y 608.45,Z 543.865,A -85,B 0,C 180,E1 -444.365,E2 -444.365} C_VEL
LIN {X 0,Y 608.432,Z 548.949,A -85,B 0,C 180,E1 -445.362,E2 -445.362} C_VEL
LIN {X 0,Y 608.449,Z 552.895,A -85,B 0,C 180,E1 -446.357,E2 -446.357} C_VEL
LIN {X 0,Y 608.425,Z 555.808,A -85,B 0,C 180,E1 -447.352,E2 -447.352} C_VEL
LIN {X 0,Y 608.444,Z 557.201,A -85,B 0,C 180,E1 -448.014,E2 -448.014} C_VEL
LIN {X 0,Y 608.439,Z 558.783,A -85,B 0,C 180,E1 -449.338,E2 -449.338} C_VEL
LIN {X 0,Y 608.434,Z 559,A -85,B 0,C 180,E1 -450,E2 -450} C_VEL
LIN {X 0,Y 608.448,Z 558.184,A -85,B 0,C 180,E1 -451.323,E2 -451.323} C_VEL
LIN {X 0,Y 608.444,Z 557.202,A -85,B 0,C 180,E1 -451.986,E2 -451.986} C_VEL
LIN {X 0,Y 608.425,Z 555.81,A -85,B 0,C 180,E1 -452.648,E2 -452.648} C_VEL
LIN {X 0,Y 608.449,Z 552.897,A -85,B 0,C 180,E1 -453.642,E2 -453.642} C_VEL
LIN {X 0,Y 608.432,Z 548.952,A -85,B 0,C 180,E1 -454.637,E2 -454.637} C_VEL
LIN {X 0,Y 608.437,Z 542.879,A -85,B 0,C 180,E1 -455.8,E2 -455.8} C_VEL
LIN {X 0,Y 608.462,Z 536.238,A -85,B 0,C 180,E1 -456.799,E2 -456.799} C_VEL
LIN {X 0,Y 608.455,Z 527.993,A -85,B 0,C 180,E1 -457.8,E2 -457.8} C_VEL
LIN {X 0,Y 608.472,Z 519.542,A -85,B 0,C 180,E1 -458.635,E2 -458.635} C_VEL
LIN {X 0,Y 608.474,Z 509.098,A -85,B 0,C 180,E1 -459.473,E2 -459.473} C_VEL
LIN {X 0,Y 608.493,Z 498.764,A -85,B 0,C 180,E1 -460.144,E2 -460.144} C_VEL
LIN {X 0,Y 608.522,Z 487.248,A -85,B 0,C 180,E1 -460.741,E2 -460.741} C_VEL
LIN {X 0,Y 608.533,Z 475.886,A -85,B 0,C 180,E1 -461.192,E2 -461.192} C_VEL
LIN {X 0,Y 608.557,Z 462.376,A -85,B 0,C 180,E1 -461.575,E2 -461.575} C_VEL
LIN {X 0,Y 608.547,Z 449.126,A -85,B 0,C 180,E1 -461.807,E2 -461.807} C_VEL
LIN {X 0,Y 608.567,Z 345.71,A -85,B 0,C 180,E1 -463.035,E2 -463.035} C_VEL
LIN {X 0,Y 608.511,Z 343.811,A -85,B 0,C 180,E1 -463.185,E2 -463.185} C_VEL
LIN {X 0,Y 608.536,Z 318.04,A -85,B 0,C 180,E1 -465.919,E2 -465.919} C_VEL
LIN {X 0,Y 608.564,Z 291.805,A -85,B 0,C 180,E1 -468.741,E2 -468.741} C_VEL
LIN {X 0,Y 608.617,Z 266.498,A -85,B 0,C 180,E1 -471.507,E2 -471.507} C_VEL
LIN {X 0,Y 608.679,Z 240.214,A -85,B 0,C 180,E1 -474.437,E2 -474.437} C_VEL
LIN {X 0,Y 608.535,Z 230.032,A -85,B 0,C 180,E1 -475.603,E2 -475.603} C_VEL
LIN {X 0,Y 608.459,Z 229.718,A -85,B 0,C 180,E1 -475.718,E2 -475.718} C_VEL
LIN {X 0,Y 608.388,Z 229.696,A -85,B 0,C 180,E1 -478.269,E2 -478.269} C_VEL
LIN {X 0,Y 608.397,Z 229.694,A -85,B 0,C 180,E1 -480.548,E2 -480.548} C_VEL
LIN {X 0,Y 608.421,Z 229.693,A -85,B 0,C 180,E1 -482.881,E2 -482.881} C_VEL
LIN {X 0,Y 608.411,Z 229.701,A -85,B 0,C 180,E1 -485.279,E2 -485.279} C_VEL
LIN {X 0,Y 608.425,Z 229.695,A -85,B 0,C 180,E1 -487.748,E2 -487.748} C_VEL
LIN {X 0,Y 608.394,Z 229.695,A -85,B 0,C 180,E1 -490.322,E2 -490.322} C_VEL
LIN {X 0,Y 608.423,Z 229.696,A -85,B 0,C 180,E1 -492.961,E2 -492.961} C_VEL
LIN {X 0,Y 608.403,Z 229.696,A -85,B 0,C 180,E1 -495.74,E2 -495.74} C_VEL
LIN {X 0,Y 608.4,Z 229.695,A -85,B 0,C 180,E1 -497.933,E2 -497.933} C_VEL
LIN {X 0,Y 608.414,Z 229.696,A -85,B 0,C 180,E1 -500.707,E2 -500.707} C_VEL
LIN {X 0,Y 608.438,Z 229.7,A -85,B 0,C 180,E1 -503.084,E2 -503.084} C_VEL
LIN {X 0,Y 608.434,Z 229.693,A -85,B 0,C 180,E1 -505.528,E2 -505.528} C_VEL
LIN {X 0,Y 608.403,Z 229.694,A -85,B 0,C 180,E1 -507.902,E2 -507.902} C_VEL
LIN {X 0,Y 608.402,Z 229.694,A -85,B 0,C 180,E1 -510.217,E2 -510.217} C_VEL
LIN {X 0,Y 608.453,Z 229.695,A -85,B 0,C 180,E1 -512.794,E2 -512.794} C_VEL
LIN {X 0,Y 608.416,Z 229.694,A -85,B 0,C 180,E1 -515.427,E2 -515.427} C_VEL
LIN {X 0,Y 608.421,Z 229.693,A -85,B 0,C 180,E1 -518.307,E2 -518.307} C_VEL
LIN {X 0,Y 608.405,Z 229.696,A -85,B 0,C 180,E1 -521.298,E2 -521.298} C_VEL
LIN {X 0,Y 608.396,Z 229.695,A -85,B 0,C 180,E1 -523.904,E2 -523.904} C_VEL
LIN {X 0,Y 608.45,Z 229.697,A -85,B 0,C 180,E1 -526.643,E2 -526.643} C_VEL
LIN {X 0,Y 608.404,Z 229.695,A -85,B 0,C 180,E1 -529.349,E2 -529.349} C_VEL
LIN {X 0,Y 608.398,Z 229.695,A -85,B 0,C 180,E1 -531.363,E2 -531.363} C_VEL
LIN {X 0,Y 608.396,Z 229.695,A -85,B 0,C 180,E1 -533.422,E2 -533.422} C_VEL
LIN {X 0,Y 608.387,Z 229.696,A -85,B 0,C 180,E1 -535.362,E2 -535.362} C_VEL
LIN {X 0,Y 608.411,Z 229.693,A -85,B 0,C 180,E1 -537.352,E2 -537.352} C_VEL
LIN {X 0,Y 608.427,Z 229.693,A -85,B 0,C 180,E1 -540,E2 -540} C_VEL
LIN {X 0,Y 608.463,Z 229.693,A -85,B 0,C 180,E1 -542.648,E2 -542.648} C_VEL
LIN {X 0,Y 608.398,Z 229.694,A -85,B 0,C 180,E1 -545.303,E2 -545.303} C_VEL
LIN {X 0,Y 608.393,Z 229.695,A -85,B 0,C 180,E1 -547.3,E2 -547.3} C_VEL
LIN {X 0,Y 608.399,Z 229.694,A -85,B 0,C 180,E1 -549.458,E2 -549.458} C_VEL
LIN {X 0,Y 607.735,Z 229.783,A -85,B 0,C 180,E1 -550.011,E2 -550.011} C_VEL
LIN {X 0,Y 604.893,Z 230.139,A -85,B 0,C 180,E1 -550.907,E2 -550.907} C_VEL
LIN {X 0,Y 602.491,Z 230.439,A -85,B 0,C 180,E1 -551.629,E2 -551.629} C_VEL
LIN {X 0,Y 601.457,Z 230.567,A -85,B 0,C 180,E1 -552.185,E2 -552.185} C_VEL
LIN {X 0,Y 601.372,Z 230.574,A -85,B 0,C 180,E1 -552.374,E2 -552.374} C_VEL
LIN {X 0,Y 601.371,Z 230.571,A -85,B 0,C 180,E1 -554.899,E2 -554.899} C_VEL
LIN {X 0,Y 601.358,Z 230.572,A -85,B 0,C 180,E1 -556.988,E2 -556.988} C_VEL
LIN {X 0,Y 601.37,Z 230.574,A -85,B 0,C 180,E1 -559.811,E2 -559.811} C_VEL
LIN {X 0,Y 601.388,Z 230.57,A -85,B 0,C 180,E1 -562.684,E2 -562.684} C_VEL
LIN {X 0,Y 601.359,Z 230.572,A -85,B 0,C 180,E1 -564.881,E2 -564.881} C_VEL
LIN {X 0,Y 601.356,Z 230.572,A -85,B 0,C 180,E1 -567.355,E2 -567.355} C_VEL
LIN {X 0,Y 601.393,Z 230.575,A -85,B 0,C 180,E1 -570.166,E2 -570.166} C_VEL
LIN {X 0,Y 601.378,Z 230.569,A -85,B 0,C 180,E1 -572.711,E2 -572.711} C_VEL
LIN {X 0,Y 601.343,Z 230.573,A -85,B 0,C 180,E1 -575.107,E2 -575.107} C_VEL
LIN {X 0,Y 601.379,Z 230.572,A -85,B 0,C 180,E1 -577.424,E2 -577.424} C_VEL
LIN {X 0,Y 601.367,Z 230.578,A -85,B 0,C 180,E1 -579.999,E2 -579.999} C_VEL
LIN {X 0,Y 601.343,Z 230.574,A -85,B 0,C 180,E1 -582.585,E2 -582.585} C_VEL
LIN {X 0,Y 601.357,Z 230.572,A -85,B 0,C 180,E1 -584.53,E2 -584.53} C_VEL
LIN {X 0,Y 601.378,Z 230.574,A -85,B 0,C 180,E1 -587.413,E2 -587.413} C_VEL
LIN {X 0,Y 601.374,Z 230.57,A -85,B 0,C 180,E1 -590.473,E2 -590.473} C_VEL
LIN {X 0,Y 601.374,Z 230.569,A -85,B 0,C 180,E1 -592.626,E2 -592.626} C_VEL
LIN {X 0,Y 601.369,Z 230.572,A -85,B 0,C 180,E1 -595.066,E2 -595.066} C_VEL
LIN {X 0,Y 601.429,Z 230.572,A -85,B 0,C 180,E1 -597.485,E2 -597.485} C_VEL
LIN {X 0,Y 601.36,Z 230.571,A -85,B 0,C 180,E1 -600.605,E2 -600.605} C_VEL
LIN {X 0,Y 601.374,Z 230.571,A -85,B 0,C 180,E1 -602.886,E2 -602.886} C_VEL
LIN {X 0,Y 601.415,Z 230.567,A -85,B 0,C 180,E1 -605.859,E2 -605.859} C_VEL
LIN {X 0,Y 601.348,Z 230.574,A -85,B 0,C 180,E1 -608.039,E2 -608.039} C_VEL
LIN {X 0,Y 601.362,Z 230.571,A -85,B 0,C 180,E1 -610.19,E2 -610.19} C_VEL
LIN {X 0,Y 601.375,Z 230.575,A -85,B 0,C 180,E1 -613.013,E2 -613.013} C_VEL
LIN {X 0,Y 601.37,Z 230.571,A -85,B 0,C 180,E1 -615.93,E2 -615.93} C_VEL
LIN {X 0,Y 601.372,Z 230.571,A -85,B 0,C 180,E1 -618.541,E2 -618.541} C_VEL
LIN {X 0,Y 601.39,Z 230.577,A -85,B 0,C 180,E1 -621.262,E2 -621.262} C_VEL
LIN {X 0,Y 601.351,Z 230.575,A -85,B 0,C 180,E1 -623.963,E2 -623.963} C_VEL
LIN {X 0,Y 601.442,Z 230.797,A -85,B 0,C 180,E1 -624.952,E2 -624.952} C_VEL
LIN {X 0,Y 601.614,Z 231.61,A -85,B 0,C 180,E1 -625.037,E2 -625.037} C_VEL
LIN {X 0,Y 601.601,Z 325.289,A -85,B 0,C 180,E1 -626.191,E2 -626.191} C_VEL
LIN {X 0,Y 601.585,Z 339,A -85,B 0,C 180,E1 -626.505,E2 -626.505} C_VEL
LIN {X 0,Y 601.555,Z 351.845,A -85,B 0,C 180,E1 -626.945,E2 -626.945} C_VEL
LIN {X 0,Y 601.508,Z 363.531,A -85,B 0,C 180,E1 -627.489,E2 -627.489} C_VEL
LIN {X 0,Y 601.462,Z 374.779,A -85,B 0,C 180,E1 -628.159,E2 -628.159} C_VEL
LIN {X 0,Y 601.458,Z 384.948,A -85,B 0,C 180,E1 -628.912,E2 -628.912} C_VEL
LIN {X 0,Y 601.415,Z 393.321,A -85,B 0,C 180,E1 -629.666,E2 -629.666} C_VEL
LIN {X 0,Y 601.393,Z 402.416,A -85,B 0,C 180,E1 -630.67,E2 -630.67} C_VEL
LIN {X 0,Y 601.36,Z 409.765,A -85,B 0,C 180,E1 -631.674,E2 -631.674} C_VEL
LIN {X 0,Y 601.342,Z 415.678,A -85,B 0,C 180,E1 -632.68,E2 -632.68} C_VEL
LIN {X 0,Y 601.367,Z 420.359,A -85,B 0,C 180,E1 -633.686,E2 -633.686} C_VEL
LIN {X 0,Y 601.329,Z 423.95,A -85,B 0,C 180,E1 -634.693,E2 -634.693} C_VEL
LIN {X 0,Y 601.349,Z 425.808,A -85,B 0,C 180,E1 -635.365,E2 -635.365} C_VEL
LIN {X 0,Y 601.35,Z 428.042,A -85,B 0,C 180,E1 -636.583,E2 -636.583} C_VEL
LIN {X 0,Y 601.322,Z 428.792,A -85,B 0,C 180,E1 -637.387,E2 -637.387} C_VEL
LIN {X 0,Y 601.333,Z 428.999,A -85,B 0,C 180,E1 -638.062,E2 -638.062} C_VEL
LIN {X 0,Y 601.336,Z 428.146,A -85,B 0,C 180,E1 -639.417,E2 -639.417} C_VEL
LIN {X 0,Y 601.33,Z 427.13,A -85,B 0,C 180,E1 -640.097,E2 -640.097} C_VEL
LIN {X 0,Y 601.337,Z 425.175,A -85,B 0,C 180,E1 -640.966,E2 -640.966} C_VEL
LIN {X 0,Y 601.367,Z 421.391,A -85,B 0,C 180,E1 -642.143,E2 -642.143} C_VEL
LIN {X 0,Y 601.348,Z 416.886,A -85,B 0,C 180,E1 -643.173,E2 -643.173} C_VEL
LIN {X 0,Y 601.384,Z 411.123,A -85,B 0,C 180,E1 -644.206,E2 -644.206} C_VEL
LIN {X 0,Y 601.38,Z 403.829,A -85,B 0,C 180,E1 -645.245,E2 -645.245} C_VEL
LIN {X 0,Y 601.407,Z 394.669,A -85,B 0,C 180,E1 -646.288,E2 -646.288} C_VEL
LIN {X 0,Y 601.447,Z 385.166,A -85,B 0,C 180,E1 -647.16,E2 -647.16} C_VEL
LIN {X 0,Y 601.487,Z 374.501,A -85,B 0,C 180,E1 -647.949,E2 -647.949} C_VEL
LIN {X 0,Y 601.529,Z 363.235,A -85,B 0,C 180,E1 -648.616,E2 -648.616} C_VEL
LIN {X 0,Y 601.561,Z 350.873,A -85,B 0,C 180,E1 -649.183,E2 -649.183} C_VEL
LIN {X 0,Y 601.579,Z 337.562,A -85,B 0,C 180,E1 -649.626,E2 -649.626} C_VEL
LIN {X 0,Y 601.634,Z 324.522,A -85,B 0,C 180,E1 -649.913,E2 -649.913} C_VEL
LIN {X 0,Y 601.672,Z 231.764,A -85,B 0,C 180,E1 -651.045,E2 -651.045} C_VEL
LIN {X 0,Y 601.448,Z 230.7,A -85,B 0,C 180,E1 -651.161,E2 -651.161} C_VEL
LIN {X 0,Y 601.427,Z 230.564,A -85,B 0,C 180,E1 -654.141,E2 -654.141} C_VEL
LIN {X 0,Y 601.423,Z 230.57,A -85,B 0,C 180,E1 -657.112,E2 -657.112} C_VEL
LIN {X 0,Y 601.38,Z 230.571,A -85,B 0,C 180,E1 -659.395,E2 -659.395} C_VEL
LIN {X 0,Y 601.39,Z 230.567,A -85,B 0,C 180,E1 -661.727,E2 -661.727} C_VEL
LIN {X 0,Y 601.411,Z 230.566,A -85,B 0,C 180,E1 -664.119,E2 -664.119} C_VEL
LIN {X 0,Y 601.389,Z 230.575,A -85,B 0,C 180,E1 -666.583,E2 -666.583} C_VEL
LIN {X 0,Y 601.382,Z 230.571,A -85,B 0,C 180,E1 -669.128,E2 -669.128} C_VEL
LIN {X 0,Y 601.406,Z 230.565,A -85,B 0,C 180,E1 -671.766,E2 -671.766} C_VEL
LIN {X 0,Y 601.396,Z 230.577,A -85,B 0,C 180,E1 -674.532,E2 -674.532} C_VEL
LIN {X 0,Y 601.36,Z 230.571,A -85,B 0,C 180,E1 -677.325,E2 -677.325} C_VEL
LIN {X 0,Y 601.396,Z 230.567,A -85,B 0,C 180,E1 -679.428,E2 -679.428} C_VEL
LIN {X 0,Y 601.397,Z 230.567,A -85,B 0,C 180,E1 -681.73,E2 -681.73} C_VEL
LIN {X 0,Y 601.381,Z 230.577,A -85,B 0,C 180,E1 -684.245,E2 -684.245} C_VEL
LIN {X 0,Y 601.402,Z 230.57,A -85,B 0,C 180,E1 -686.684,E2 -686.684} C_VEL
LIN {X 0,Y 601.385,Z 230.567,A -85,B 0,C 180,E1 -689.056,E2 -689.056} C_VEL
LIN {X 0,Y 601.394,Z 230.567,A -85,B 0,C 180,E1 -691.371,E2 -691.371} C_VEL
LIN {X 0,Y 601.4,Z 230.572,A -85,B 0,C 180,E1 -694.381,E2 -694.381} C_VEL
LIN {X 0,Y 601.375,Z 230.571,A -85,B 0,C 180,E1 -696.588,E2 -696.588} C_VEL
LIN {X 0,Y 601.406,Z 230.566,A -85,B 0,C 180,E1 -699.477,E2 -699.477} C_VEL
LIN {X 0,Y 601.372,Z 230.575,A -85,B 0,C 180,E1 -702.311,E2 -702.311} C_VEL
LIN {X 0,Y 601.383,Z 230.571,A -85,B 0,C 180,E1 -704.408,E2 -704.408} C_VEL
LIN {X 0,Y 601.389,Z 230.568,A -85,B 0,C 180,E1 -707.171,E2 -707.171} C_VEL
LIN {X 0,Y 601.411,Z 230.574,A -85,B 0,C 180,E1 -709.904,E2 -709.904} C_VEL
LIN {X 0,Y 601.363,Z 230.571,A -85,B 0,C 180,E1 -712.614,E2 -712.614} C_VEL
LIN {X 0,Y 601.403,Z 230.569,A -85,B 0,C 180,E1 -715.308,E2 -715.308} C_VEL
LIN {X 0,Y 601.399,Z 230.572,A -85,B 0,C 180,E1 -717.991,E2 -717.991} C_VEL
LIN {X 0,Y 601.418,Z 230.568,A -85,B 0,C 180,E1 -720,E2 -720} C_VEL
LIN {X 0,Y 601.391,Z 230.567,A -85,B 0,C 180,E1 -722.679,E2 -722.679} C_VEL
LIN {X 0,Y 601.413,Z 230.571,A -85,B 0,C 180,E1 -725.364,E2 -725.364} C_VEL
LIN {X 0,Y 601.386,Z 230.57,A -85,B 0,C 180,E1 -728.061,E2 -728.061} C_VEL
LIN {X 0,Y 601.374,Z 230.57,A -85,B 0,C 180,E1 -730.777,E2 -730.777} C_VEL
LIN {X 0,Y 601.398,Z 230.575,A -85,B 0,C 180,E1 -733.516,E2 -733.516} C_VEL
LIN {X 0,Y 601.379,Z 230.569,A -85,B 0,C 180,E1 -736.289,E2 -736.289} C_VEL
LIN {X 0,Y 601.398,Z 230.573,A -85,B 0,C 180,E1 -739.1,E2 -739.1} C_VEL
LIN {X 0,Y 601.382,Z 230.579,A -85,B 0,C 180,E1 -741.24,E2 -741.24} C_VEL
LIN {X 0,Y 601.365,Z 230.578,A -85,B 0,C 180,E1 -743.413,E2 -743.413} C_VEL
LIN {X 0,Y 601.368,Z 230.571,A -85,B 0,C 180,E1 -745.861,E2 -745.861} C_VEL
LIN {X 0,Y 601.351,Z 230.572,A -85,B 0,C 180,E1 -747.871,E2 -747.871} C_VEL
LIN {X 0,Y 601.363,Z 230.571,A -85,B 0,C 180,E1 -750.168,E2 -750.168} C_VEL
LIN {X 0,Y 601.387,Z 230.572,A -85,B 0,C 180,E1 -752.712,E2 -752.712} C_VEL
LIN {X 0,Y 601.378,Z 230.577,A -85,B 0,C 180,E1 -755.111,E2 -755.111} C_VEL
LIN {X 0,Y 601.386,Z 230.571,A -85,B 0,C 180,E1 -757.423,E2 -757.423} C_VEL
LIN {X 0,Y 601.366,Z 230.57,A -85,B 0,C 180,E1 -759.999,E2 -759.999} C_VEL
LIN {X 0,Y 601.367,Z 230.578,A -85,B 0,C 180,E1 -762.674,E2 -762.674} C_VEL
LIN {X 0,Y 601.36,Z 230.572,A -85,B 0,C 180,E1 -765.477,E2 -765.477} C_VEL
LIN {X 0,Y 601.39,Z 230.57,A -85,B 0,C 180,E1 -768.233,E2 -768.233} C_VEL
LIN {X 0,Y 601.381,Z 230.576,A -85,B 0,C 180,E1 -770.872,E2 -770.872} C_VEL
LIN {X 0,Y 601.366,Z 230.571,A -85,B 0,C 180,E1 -773.415,E2 -773.415} C_VEL
LIN {X 0,Y 601.406,Z 230.568,A -85,B 0,C 180,E1 -776.068,E2 -776.068} C_VEL
LIN {X 0,Y 601.379,Z 230.572,A -85,B 0,C 180,E1 -779.056,E2 -779.056} C_VEL
LIN {X 0,Y 601.349,Z 230.573,A -85,B 0,C 180,E1 -781.369,E2 -781.369} C_VEL
LIN {X 0,Y 601.429,Z 230.697,A -85,B 0,C 180,E1 -784.13,E2 -784.13} C_VEL
LIN {X 0,Y 601.92,Z 234.279,A -85,B 0,C 180,E1 -784.59,E2 -784.59} C_VEL
LIN {X 0,Y 601.783,Z 256.991,A -85,B 0,C 180,E1 -787.169,E2 -787.169} C_VEL
LIN {X 0,Y 601.686,Z 280.989,A -85,B 0,C 180,E1 -789.844,E2 -789.844} C_VEL
LIN {X 0,Y 601.606,Z 306.76,A -85,B 0,C 180,E1 -792.669,E2 -792.669} C_VEL
LIN {X 0,Y 601.541,Z 332.531,A -85,B 0,C 180,E1 -795.452,E2 -795.452} C_VEL
LIN {X 0,Y 601.52,Z 345.155,A -85,B 0,C 180,E1 -796.788,E2 -796.788} C_VEL
LIN {X 0,Y 601.67,Z 350.721,A -85,B 0,C 180,E1 -796.877,E2 -796.877} C_VEL
LIN {X 0,Y 601.608,Z 454.946,A -85,B 0,C 180,E1 -798.139,E2 -798.139} C_VEL
LIN {X 0,Y 601.588,Z 468.216,A -85,B 0,C 180,E1 -798.438,E2 -798.438} C_VEL
LIN {X 0,Y 601.549,Z 479.922,A -85,B 0,C 180,E1 -798.826,E2 -798.826} C_VEL
LIN {X 0,Y 601.516,Z 490.923,A -85,B 0,C 180,E1 -799.311,E2 -799.311} C_VEL
LIN {X 0,Y 601.478,Z 501.579,A -85,B 0,C 180,E1 -799.906,E2 -799.906} C_VEL
LIN {X 0,Y 601.447,Z 512.475,A -85,B 0,C 180,E1 -800.669,E2 -800.669} C_VEL
LIN {X 0,Y 601.429,Z 523.111,A -85,B 0,C 180,E1 -801.601,E2 -801.601} C_VEL
LIN {X 0,Y 601.418,Z 530.959,A -85,B 0,C 180,E1 -802.446,E2 -802.446} C_VEL
LIN {X 0,Y 601.37,Z 538.224,A -85,B 0,C 180,E1 -803.398,E2 -803.398} C_VEL
LIN {X 0,Y 601.372,Z 543.865,A -85,B 0,C 180,E1 -804.299,E2 -804.299} C_VEL
LIN {X 0,Y 601.336,Z 548.949,A -85,B 0,C 180,E1 -805.307,E2 -805.307} C_VEL
LIN {X 0,Y 601.367,Z 552.895,A -85,B 0,C 180,E1 -806.314,E2 -806.314} C_VEL
LIN {X 0,Y 601.325,Z 555.808,A -85,B 0,C 180,E1 -807.32,E2 -807.32} C_VEL
LIN {X 0,Y 601.343,Z 557.201,A -85,B 0,C 180,E1 -807.99,E2 -807.99} C_VEL
LIN {X 0,Y 601.339,Z 558.784,A -85,B 0,C 180,E1 -809.33,E2 -809.33} C_VEL
LIN {X 0,Y 601.335,Z 559,A -85,B 0,C 180,E1 -810,E2 -810} C_VEL
LIN {X 0,Y 601.348,Z 558.185,A -85,B 0,C 180,E1 -811.339,E2 -811.339} C_VEL
LIN {X 0,Y 601.343,Z 557.202,A -85,B 0,C 180,E1 -812.009,E2 -812.009} C_VEL
LIN {X 0,Y 601.325,Z 555.81,A -85,B 0,C 180,E1 -812.679,E2 -812.679} C_VEL
LIN {X 0,Y 601.367,Z 552.897,A -85,B 0,C 180,E1 -813.685,E2 -813.685} C_VEL
LIN {X 0,Y 601.336,Z 548.951,A -85,B 0,C 180,E1 -814.692,E2 -814.692} C_VEL
LIN {X 0,Y 601.372,Z 542.88,A -85,B 0,C 180,E1 -815.869,E2 -815.869} C_VEL
LIN {X 0,Y 601.381,Z 536.239,A -85,B 0,C 180,E1 -816.879,E2 -816.879} C_VEL
LIN {X 0,Y 601.4,Z 527.993,A -85,B 0,C 180,E1 -817.892,E2 -817.892} C_VEL
LIN {X 0,Y 601.436,Z 519.542,A -85,B 0,C 180,E1 -818.737,E2 -818.737} C_VEL
LIN {X 0,Y 601.446,Z 509.099,A -85,B 0,C 180,E1 -819.585,E2 -819.585} C_VEL
LIN {X 0,Y 601.471,Z 498.766,A -85,B 0,C 180,E1 -820.264,E2 -820.264} C_VEL
LIN {X 0,Y 601.537,Z 487.902,A -85,B 0,C 180,E1 -820.836,E2 -820.836} C_VEL
LIN {X 0,Y 601.565,Z 475.387,A -85,B 0,C 180,E1 -821.34,E2 -821.34} C_VEL
LIN {X 0,Y 601.601,Z 462.375,A -85,B 0,C 180,E1 -821.711,E2 -821.711} C_VEL
LIN {X 0,Y 601.617,Z 449.126,A -85,B 0,C 180,E1 -821.945,E2 -821.945} C_VEL
LIN {X 0,Y 601.56,Z 345.699,A -85,B 0,C 180,E1 -823.19,E2 -823.19} C_VEL
LIN {X 0,Y 601.485,Z 343.811,A -85,B 0,C 180,E1 -823.342,E2 -823.342} C_VEL
LIN {X 0,Y 601.568,Z 318.04,A -85,B 0,C 180,E1 -826.108,E2 -826.108} C_VEL
LIN {X 0,Y 601.655,Z 292.532,A -85,B 0,C 180,E1 -828.885,E2 -828.885} C_VEL
LIN {X 0,Y 601.753,Z 266.498,A -85,B 0,C 180,E1 -831.765,E2 -831.765} C_VEL
LIN {X 0,Y 601.899,Z 240.437,A -85,B 0,C 180,E1 -834.705,E2 -834.705} C_VEL
LIN {X 0,Y 601.86,Z 232.674,A -85,B 0,C 180,E1 -835.597,E2 -835.597} C_VEL
LIN {X 0,Y 601.424,Z 230.701,A -85,B 0,C 180,E1 -835.869,E2 -835.869} C_VEL
LIN {X 0,Y 601.363,Z 230.572,A -85,B 0,C 180,E1 -838.776,E2 -838.776} C_VEL
LIN {X 0,Y 601.373,Z 230.576,A -85,B 0,C 180,E1 -841.727,E2 -841.727} C_VEL
LIN {X 0,Y 601.393,Z 230.568,A -85,B 0,C 180,E1 -844.119,E2 -844.119} C_VEL
LIN {X 0,Y 601.362,Z 230.571,A -85,B 0,C 180,E1 -846.585,E2 -846.585} C_VEL
LIN {X 0,Y 601.383,Z 230.575,A -85,B 0,C 180,E1 -849.529,E2 -849.529} C_VEL
LIN {X 0,Y 601.387,Z 230.571,A -85,B 0,C 180,E1 -851.767,E2 -851.767} C_VEL
LIN {X 0,Y 601.355,Z 230.572,A -85,B 0,C 180,E1 -854.528,E2 -854.528} C_VEL
LIN {X 0,Y 601.362,Z 230.579,A -85,B 0,C 180,E1 -857.325,E2 -857.325} C_VEL
LIN {X 0,Y 601.361,Z 230.571,A -85,B 0,C 180,E1 -860.001,E2 -860.001} C_VEL
LIN {X 0,Y 601.384,Z 230.571,A -85,B 0,C 180,E1 -862.622,E2 -862.622} C_VEL
LIN {X 0,Y 601.391,Z 230.567,A -85,B 0,C 180,E1 -865.879,E2 -865.879} C_VEL
LIN {X 0,Y 601.376,Z 230.572,A -85,B 0,C 180,E1 -868.55,E2 -868.55} C_VEL
LIN {X 0,Y 601.389,Z 230.571,A -85,B 0,C 180,E1 -871.371,E2 -871.371} C_VEL
LIN {X 0,Y 601.365,Z 230.571,A -85,B 0,C 180,E1 -873.634,E2 -873.634} C_VEL
LIN {X 0,Y 601.372,Z 230.569,A -85,B 0,C 180,E1 -875.856,E2 -875.856} C_VEL
LIN {X 0,Y 601.357,Z 230.572,A -85,B 0,C 180,E1 -878.039,E2 -878.039} C_VEL
LIN {X 0,Y 601.365,Z 230.572,A -85,B 0,C 180,E1 -880.189,E2 -880.189} C_VEL
LIN {X 0,Y 601.387,Z 230.574,A -85,B 0,C 180,E1 -883.013,E2 -883.013} C_VEL
LIN {X 0,Y 601.36,Z 230.571,A -85,B 0,C 180,E1 -885.793,E2 -885.793} C_VEL
LIN {X 0,Y 601.412,Z 230.572,A -85,B 0,C 180,E1 -888.542,E2 -888.542} C_VEL
LIN {X 0,Y 601.368,Z 230.572,A -85,B 0,C 180,E1 -891.261,E2 -891.261} C_VEL
LIN {X 0,Y 601.367,Z 230.571,A -85,B 0,C 180,E1 -893.385,E2 -893.385} C_VEL
LIN {X 0,Y 601.363,Z 230.571,A -85,B 0,C 180,E1 -895.308,E2 -895.308} C_VEL
LIN {X 0,Y 601.383,Z 230.569,A -85,B 0,C 180,E1 -897.321,E2 -897.321} C_VEL
LIN {X 0,Y 601.399,Z 230.569,A -85,B 0,C 180,E1 -900,E2 -900} C_VEL
LIN {X 0,Y 601.424,Z 230.57,A -85,B 0,C 180,E1 -902.679,E2 -902.679} C_VEL
LIN {X 0,Y 601.366,Z 230.57,A -85,B 0,C 180,E1 -905.365,E2 -905.365} C_VEL
LIN {X 0,Y 601.348,Z 230.572,A -85,B 0,C 180,E1 -907.386,E2 -907.386} C_VEL
LIN {X 0,Y 601.376,Z 230.575,A -85,B 0,C 180,E1 -910.096,E2 -910.096} C_VEL
LIN {X 0,Y 601.372,Z 230.574,A -85,B 0,C 180,E1 -912.374,E2 -912.374} C_VEL
LIN {X 0,Y 600.702,Z 230.655,A -85,B 0,C 180,E1 -912.933,E2 -912.933} C_VEL
LIN {X 0,Y 597.845,Z 231.012,A -85,B 0,C 180,E1 -913.841,E2 -913.841} C_VEL
LIN {X 0,Y 595.433,Z 231.315,A -85,B 0,C 180,E1 -914.571,E2 -914.571} C_VEL
LIN {X 0,Y 594.397,Z 231.439,A -85,B 0,C 180,E1 -915.135,E2 -915.135} C_VEL
LIN {X 0,Y 594.312,Z 231.449,A -85,B 0,C 180,E1 -915.325,E2 -915.325} C_VEL
LIN {X 0,Y 594.308,Z 231.449,A -85,B 0,C 180,E1 -917.196,E2 -917.196} C_VEL
LIN {X 0,Y 594.342,Z 231.454,A -85,B 0,C 180,E1 -920.055,E2 -920.055} C_VEL
LIN {X 0,Y 594.332,Z 231.447,A -85,B 0,C 180,E1 -922.969,E2 -922.969} C_VEL
LIN {X 0,Y 594.309,Z 231.449,A -85,B 0,C 180,E1 -925.196,E2 -925.196} C_VEL
LIN {X 0,Y 594.33,Z 231.449,A -85,B 0,C 180,E1 -927.519,E2 -927.519} C_VEL
LIN {X 0,Y 594.349,Z 231.446,A -85,B 0,C 180,E1 -930.562,E2 -930.562} C_VEL
LIN {X 0,Y 594.325,Z 231.447,A -85,B 0,C 180,E1 -932.954,E2 -932.954} C_VEL
LIN {X 0,Y 594.3,Z 231.453,A -85,B 0,C 180,E1 -935.413,E2 -935.413} C_VEL
LIN {X 0,Y 594.337,Z 231.455,A -85,B 0,C 180,E1 -937.945,E2 -937.945} C_VEL
LIN {X 0,Y 594.32,Z 231.448,A -85,B 0,C 180,E1 -940.818,E2 -940.818} C_VEL
LIN {X 0,Y 594.327,Z 231.45,A -85,B 0,C 180,E1 -943.304,E2 -943.304} C_VEL
LIN {X 0,Y 594.334,Z 231.45,A -85,B 0,C 180,E1 -946.165,E2 -946.165} C_VEL
LIN {X 0,Y 594.342,Z 231.446,A -85,B 0,C 180,E1 -948.534,E2 -948.534} C_VEL
LIN {X 0,Y 594.351,Z 231.448,A -85,B 0,C 180,E1 -951.3,E2 -951.3} C_VEL
LIN {X 0,Y 594.333,Z 231.454,A -85,B 0,C 180,E1 -953.756,E2 -953.756} C_VEL
LIN {X 0,Y 594.314,Z 231.45,A -85,B 0,C 180,E1 -956.236,E2 -956.236} C_VEL
LIN {X 0,Y 594.307,Z 231.45,A -85,B 0,C 180,E1 -958.647,E2 -958.647} C_VEL
LIN {X 0,Y 594.372,Z 231.445,A -85,B 0,C 180,E1 -961.045,E2 -961.045} C_VEL
LIN {X 0,Y 594.338,Z 231.447,A -85,B 0,C 180,E1 -964.055,E2 -964.055} C_VEL
LIN {X 0,Y 594.338,Z 231.446,A -85,B 0,C 180,E1 -966.295,E2 -966.295} C_VEL
LIN {X 0,Y 594.395,Z 231.447,A -85,B 0,C 180,E1 -969.225,E2 -969.225} C_VEL
LIN {X 0,Y 594.31,Z 231.45,A -85,B 0,C 180,E1 -972.094,E2 -972.094} C_VEL
LIN {X 0,Y 594.321,Z 231.448,A -85,B 0,C 180,E1 -974.218,E2 -974.218} C_VEL
LIN {X 0,Y 594.333,Z 231.453,A -85,B 0,C 180,E1 -977.017,E2 -977.017} C_VEL
LIN {X 0,Y 594.368,Z 231.451,A -85,B 0,C 180,E1 -979.095,E2 -979.095} C_VEL
LIN {X 0,Y 594.31,Z 231.452,A -85,B 0,C 180,E1 -981.842,E2 -981.842} C_VEL
LIN {X 0,Y 594.355,Z 231.449,A -85,B 0,C 180,E1 -984.572,E2 -984.572} C_VEL
LIN {X 0,Y 594.406,Z 231.684,A -85,B 0,C 180,E1 -984.807,E2 -984.807} C_VEL
LIN {X 0,Y 594.659,Z 232.764,A -85,B 0,C 180,E1 -984.904,E2 -984.904} C_VEL
LIN {X 0,Y 594.676,Z 324.735,A -85,B 0,C 180,E1 -986.04,E2 -986.04} C_VEL
LIN {X 0,Y 594.632,Z 337.9,A -85,B 0,C 180,E1 -986.337,E2 -986.337} C_VEL
LIN {X 0,Y 594.582,Z 351.053,A -85,B 0,C 180,E1 -986.782,E2 -986.782} C_VEL
LIN {X 0,Y 594.516,Z 362.166,A -85,B 0,C 180,E1 -987.29,E2 -987.29} C_VEL
LIN {X 0,Y 594.448,Z 373.691,A -85,B 0,C 180,E1 -987.968,E2 -987.968} C_VEL
LIN {X 0,Y 594.435,Z 385.089,A -85,B 0,C 180,E1 -988.815,E2 -988.815} C_VEL
LIN {X 0,Y 594.363,Z 394.265,A -85,B 0,C 180,E1 -989.662,E2 -989.662} C_VEL
LIN {X 0,Y 594.341,Z 403.18,A -85,B 0,C 180,E1 -990.678,E2 -990.678} C_VEL
LIN {X 0,Y 594.283,Z 410.395,A -85,B 0,C 180,E1 -991.694,E2 -991.694} C_VEL
LIN {X 0,Y 594.253,Z 416.188,A -85,B 0,C 180,E1 -992.712,E2 -992.712} C_VEL
LIN {X 0,Y 594.289,Z 420.76,A -85,B 0,C 180,E1 -993.729,E2 -993.729} C_VEL
LIN {X 0,Y 594.23,Z 424.251,A -85,B 0,C 180,E1 -994.749,E2 -994.749} C_VEL
LIN {X 0,Y 594.263,Z 426.025,A -85,B 0,C 180,E1 -995.429,E2 -995.429} C_VEL
LIN {X 0,Y 594.272,Z 428.303,A -85,B 0,C 180,E1 -996.792,E2 -996.792} C_VEL
LIN {X 0,Y 594.248,Z 428.858,A -85,B 0,C 180,E1 -997.475,E2 -997.475} C_VEL
LIN {X 0,Y 594.229,Z 428.98,A -85,B 0,C 180,E1 -998.159,E2 -998.159} C_VEL
LIN {X 0,Y 594.256,Z 428.034,A -85,B 0,C 180,E1 -999.531,E2 -999.531} C_VEL
LIN {X 0,Y 594.231,Z 426.957,A -85,B 0,C 180,E1 -1000.219,E2 -1000.219} C_VEL
LIN {X 0,Y 594.252,Z 425.169,A -85,B 0,C 180,E1 -1001.003,E2 -1001.003} C_VEL
LIN {X 0,Y 594.258,Z 421.031,A -85,B 0,C 180,E1 -1002.291,E2 -1002.291} C_VEL
LIN {X 0,Y 594.274,Z 416.416,A -85,B 0,C 180,E1 -1003.333,E2 -1003.333} C_VEL
LIN {X 0,Y 594.307,Z 410.502,A -85,B 0,C 180,E1 -1004.379,E2 -1004.379} C_VEL
LIN {X 0,Y 594.34,Z 403.039,A -85,B 0,C 180,E1 -1005.43,E2 -1005.43} C_VEL
LIN {X 0,Y 594.364,Z 393.71,A -85,B 0,C 180,E1 -1006.486,E2 -1006.486} C_VEL
LIN {X 0,Y 594.431,Z 383.927,A -85,B 0,C 180,E1 -1007.369,E2 -1007.369} C_VEL
LIN {X 0,Y 594.468,Z 372.992,A -85,B 0,C 180,E1 -1008.168,E2 -1008.168} C_VEL
LIN {X 0,Y 594.544,Z 362.265,A -85,B 0,C 180,E1 -1008.794,E2 -1008.794} C_VEL
LIN {X 0,Y 594.58,Z 349.398,A -85,B 0,C 180,E1 -1009.372,E2 -1009.372} C_VEL
LIN {X 0,Y 594.642,Z 336.361,A -85,B 0,C 180,E1 -1009.797,E2 -1009.797} C_VEL
LIN {X 0,Y 594.7,Z 323.777,A -85,B 0,C 180,E1 -1010.065,E2 -1010.065} C_VEL
LIN {X 0,Y 594.701,Z 232.925,A -85,B 0,C 180,E1 -1011.18,E2 -1011.18} C_VEL
LIN {X 0,Y 594.427,Z 231.72,A -85,B 0,C 180,E1 -1011.276,E2 -1011.276} C_VEL
LIN {X 0,Y 594.366,Z 231.448,A -85,B 0,C 180,E1 -1011.503,E2 -1011.503} C_VEL
LIN {X 0,Y 594.37,Z 231.446,A -85,B 0,C 180,E1 -1014.447,E2 -1014.447} C_VEL
LIN {X 0,Y 594.345,Z 231.447,A -85,B 0,C 180,E1 -1017.518,E2 -1017.518} C_VEL
LIN {X 0,Y 594.349,Z 231.445,A -85,B 0,C 180,E1 -1019.777,E2 -1019.777} C_VEL
LIN {X 0,Y 594.364,Z 231.443,A -85,B 0,C 180,E1 -1022.147,E2 -1022.147} C_VEL
LIN {X 0,Y 594.372,Z 231.45,A -85,B 0,C 180,E1 -1024.58,E2 -1024.58} C_VEL
LIN {X 0,Y 594.353,Z 231.443,A -85,B 0,C 180,E1 -1027.603,E2 -1027.603} C_VEL
LIN {X 0,Y 594.356,Z 231.454,A -85,B 0,C 180,E1 -1030.567,E2 -1030.567} C_VEL
LIN {X 0,Y 594.346,Z 231.446,A -85,B 0,C 180,E1 -1033.301,E2 -1033.301} C_VEL
LIN {X 0,Y 594.342,Z 231.45,A -85,B 0,C 180,E1 -1036.162,E2 -1036.162} C_VEL
LIN {X 0,Y 594.368,Z 231.451,A -85,B 0,C 180,E1 -1038.535,E2 -1038.535} C_VEL
LIN {X 0,Y 594.358,Z 231.443,A -85,B 0,C 180,E1 -1041.298,E2 -1041.298} C_VEL
LIN {X 0,Y 594.34,Z 231.446,A -85,B 0,C 180,E1 -1043.754,E2 -1043.754} C_VEL
LIN {X 0,Y 594.366,Z 231.452,A -85,B 0,C 180,E1 -1046.238,E2 -1046.238} C_VEL
LIN {X 0,Y 594.354,Z 231.446,A -85,B 0,C 180,E1 -1048.648,E2 -1048.648} C_VEL
LIN {X 0,Y 594.366,Z 231.442,A -85,B 0,C 180,E1 -1051.044,E2 -1051.044} C_VEL
LIN {X 0,Y 594.357,Z 231.452,A -85,B 0,C 180,E1 -1054.055,E2 -1054.055} C_VEL
LIN {X 0,Y 594.366,Z 231.448,A -85,B 0,C 180,E1 -1056.295,E2 -1056.295} C_VEL
LIN {X 0,Y 594.376,Z 231.439,A -85,B 0,C 180,E1 -1059.223,E2 -1059.223} C_VEL
LIN {X 0,Y 594.331,Z 231.456,A -85,B 0,C 180,E1 -1062.094,E2 -1062.094} C_VEL
LIN {X 0,Y 594.339,Z 231.451,A -85,B 0,C 180,E1 -1064.218,E2 -1064.218} C_VEL
LIN {X 0,Y 594.356,Z 231.447,A -85,B 0,C 180,E1 -1066.32,E2 -1066.32} C_VEL
LIN {X 0,Y 594.336,Z 231.446,A -85,B 0,C 180,E1 -1069.094,E2 -1069.094} C_VEL
LIN {X 0,Y 594.366,Z 231.453,A -85,B 0,C 180,E1 -1071.842,E2 -1071.842} C_VEL
LIN {X 0,Y 594.348,Z 231.445,A -85,B 0,C 180,E1 -1074.572,E2 -1074.572} C_VEL
LIN {X 0,Y 594.39,Z 231.442,A -85,B 0,C 180,E1 -1077.289,E2 -1077.289} C_VEL
LIN {X 0,Y 594.388,Z 231.444,A -85,B 0,C 180,E1 -1080,E2 -1080} C_VEL
LIN {X 0,Y 594.362,Z 231.442,A -85,B 0,C 180,E1 -1082.711,E2 -1082.711} C_VEL
LIN {X 0,Y 594.375,Z 231.449,A -85,B 0,C 180,E1 -1085.428,E2 -1085.428} C_VEL
LIN {X 0,Y 594.339,Z 231.447,A -85,B 0,C 180,E1 -1088.158,E2 -1088.158} C_VEL
LIN {X 0,Y 594.359,Z 231.447,A -85,B 0,C 180,E1 -1091.063,E2 -1091.063} C_VEL
LIN {X 0,Y 594.32,Z 231.448,A -85,B 0,C 180,E1 -1094.151,E2 -1094.151} C_VEL
LIN {X 0,Y 594.362,Z 231.451,A -85,B 0,C 180,E1 -1097.194,E2 -1097.194} C_VEL
LIN {X 0,Y 594.341,Z 231.446,A -85,B 0,C 180,E1 -1100.055,E2 -1100.055} C_VEL
LIN {X 0,Y 594.336,Z 231.452,A -85,B 0,C 180,E1 -1102.968,E2 -1102.968} C_VEL
LIN {X 0,Y 594.33,Z 231.447,A -85,B 0,C 180,E1 -1105.946,E2 -1105.946} C_VEL
LIN {X 0,Y 594.313,Z 231.448,A -85,B 0,C 180,E1 -1108.23,E2 -1108.23} C_VEL
LIN {X 0,Y 594.345,Z 231.447,A -85,B 0,C 180,E1 -1110.562,E2 -1110.562} C_VEL
LIN {X 0,Y 594.36,Z 231.452,A -85,B 0,C 180,E1 -1112.951,E2 -1112.951} C_VEL
LIN {X 0,Y 594.31,Z 231.453,A -85,B 0,C 180,E1 -1115.412,E2 -1115.412} C_VEL
LIN {X 0,Y 594.345,Z 231.445,A -85,B 0,C 180,E1 -1117.944,E2 -1117.944} C_VEL
LIN {X 0,Y 594.357,Z 231.453,A -85,B 0,C 180,E1 -1120.821,E2 -1120.821} C_VEL
LIN {X 0,Y 594.334,Z 231.446,A -85,B 0,C 180,E1 -1123.837,E2 -1123.837} C_VEL
LIN {X 0,Y 594.336,Z 231.455,A -85,B 0,C 180,E1 -1126.699,E2 -1126.699} C_VEL
LIN {X 0,Y 594.334,Z 231.447,A -85,B 0,C 180,E1 -1129.431,E2 -1129.431} C_VEL
LIN {X 0,Y 594.35,Z 231.45,A -85,B 0,C 180,E1 -1132.397,E2 -1132.397} C_VEL
LIN {X 0,Y 594.346,Z 231.445,A -85,B 0,C 180,E1 -1135.418,E2 -1135.418} C_VEL
LIN {X 0,Y 594.351,Z 231.451,A -85,B 0,C 180,E1 -1138.362,E2 -1138.362} C_VEL
LIN {X 0,Y 594.329,Z 231.45,A -85,B 0,C 180,E1 -1141.052,E2 -1141.052} C_VEL
LIN {X 0,Y 594.383,Z 231.601,A -85,B 0,C 180,E1 -1143.916,E2 -1143.916} C_VEL
LIN {X 0,Y 595.128,Z 235.89,A -85,B 0,C 180,E1 -1144.467,E2 -1144.467} C_VEL
LIN {X 0,Y 594.947,Z 259.099,A -85,B 0,C 180,E1 -1147.132,E2 -1147.132} C_VEL
LIN {X 0,Y 594.802,Z 282.6,A -85,B 0,C 180,E1 -1149.781,E2 -1149.781} C_VEL
LIN {X 0,Y 594.658,Z 308.371,A -85,B 0,C 180,E1 -1152.637,E2 -1152.637} C_VEL
LIN {X 0,Y 594.527,Z 334.142,A -85,B 0,C 180,E1 -1155.452,E2 -1155.452} C_VEL
LIN {X 0,Y 594.511,Z 345.151,A -85,B 0,C 180,E1 -1156.629,E2 -1156.629} C_VEL
LIN {X 0,Y 594.782,Z 348.932,A -85,B 0,C 180,E1 -1156.7,E2 -1156.7} C_VEL
LIN {X 0,Y 594.66,Z 454.946,A -85,B 0,C 180,E1 -1157.999,E2 -1157.999} C_VEL
LIN {X 0,Y 594.635,Z 468.217,A -85,B 0,C 180,E1 -1158.301,E2 -1158.301} C_VEL
LIN {X 0,Y 594.595,Z 480.575,A -85,B 0,C 180,E1 -1158.719,E2 -1158.719} C_VEL
LIN {X 0,Y 594.539,Z 492.631,A -85,B 0,C 180,E1 -1159.27,E2 -1159.27} C_VEL
LIN {X 0,Y 594.48,Z 504.199,A -85,B 0,C 180,E1 -1159.958,E2 -1159.958} C_VEL
LIN {X 0,Y 594.413,Z 514.596,A -85,B 0,C 180,E1 -1160.73,E2 -1160.73} C_VEL
LIN {X 0,Y 594.383,Z 523.111,A -85,B 0,C 180,E1 -1161.5,E2 -1161.5} C_VEL
LIN {X 0,Y 594.347,Z 530.959,A -85,B 0,C 180,E1 -1162.355,E2 -1162.355} C_VEL
LIN {X 0,Y 594.283,Z 538.812,A -85,B 0,C 180,E1 -1163.408,E2 -1163.408} C_VEL
LIN {X 0,Y 594.289,Z 545.679,A -85,B 0,C 180,E1 -1164.571,E2 -1164.571} C_VEL
LIN {X 0,Y 594.27,Z 550.371,A -85,B 0,C 180,E1 -1165.591,E2 -1165.591} C_VEL
LIN {X 0,Y 594.267,Z 553.956,A -85,B 0,C 180,E1 -1166.61,E2 -1166.61} C_VEL
LIN {X 0,Y 594.226,Z 555.808,A -85,B 0,C 180,E1 -1167.288,E2 -1167.288} C_VEL
LIN {X 0,Y 594.242,Z 557.201,A -85,B 0,C 180,E1 -1167.966,E2 -1167.966} C_VEL
LIN {X 0,Y 594.239,Z 558.784,A -85,B 0,C 180,E1 -1169.322,E2 -1169.322} C_VEL
LIN {X 0,Y 594.236,Z 559,A -85,B 0,C 180,E1 -1170,E2 -1170} C_VEL
LIN {X 0,Y 594.248,Z 558.185,A -85,B 0,C 180,E1 -1171.355,E2 -1171.355} C_VEL
LIN {X 0,Y 594.242,Z 557.202,A -85,B 0,C 180,E1 -1172.033,E2 -1172.033} C_VEL
LIN {X 0,Y 594.226,Z 555.81,A -85,B 0,C 180,E1 -1172.711,E2 -1172.711} C_VEL
LIN {X 0,Y 594.288,Z 552.897,A -85,B 0,C 180,E1 -1173.729,E2 -1173.729} C_VEL
LIN {X 0,Y 594.241,Z 548.951,A -85,B 0,C 180,E1 -1174.748,E2 -1174.748} C_VEL
LIN {X 0,Y 594.304,Z 542.88,A -85,B 0,C 180,E1 -1175.939,E2 -1175.939} C_VEL
LIN {X 0,Y 594.307,Z 536.239,A -85,B 0,C 180,E1 -1176.962,E2 -1176.962} C_VEL
LIN {X 0,Y 594.359,Z 527.994,A -85,B 0,C 180,E1 -1177.986,E2 -1177.986} C_VEL
LIN {X 0,Y 594.382,Z 519.543,A -85,B 0,C 180,E1 -1178.842,E2 -1178.842} C_VEL
LIN {X 0,Y 594.427,Z 509.101,A -85,B 0,C 180,E1 -1179.699,E2 -1179.699} C_VEL
LIN {X 0,Y 594.484,Z 498.768,A -85,B 0,C 180,E1 -1180.386,E2 -1180.386} C_VEL
LIN {X 0,Y 594.561,Z 487.692,A -85,B 0,C 180,E1 -1180.975,E2 -1180.975} C_VEL
LIN {X 0,Y 594.6,Z 475.715,A -85,B 0,C 180,E1 -1181.464,E2 -1181.464} C_VEL
LIN {X 0,Y 594.643,Z 462.374,A -85,B 0,C 180,E1 -1181.85,E2 -1181.85} C_VEL
LIN {X 0,Y 594.691,Z 449.126,A -85,B 0,C 180,E1 -1182.087,E2 -1182.087} C_VEL
LIN {X 0,Y 594.667,Z 346.521,A -85,B 0,C 180,E1 -1183.332,E2 -1183.332} C_VEL
LIN {X 0,Y 594.49,Z 344.861,A -85,B 0,C 180,E1 -1183.393,E2 -1183.393} C_VEL
LIN {X 0,Y 594.604,Z 319.651,A -85,B 0,C 180,E1 -1186.126,E2 -1186.126} C_VEL
LIN {X 0,Y 594.743,Z 294.447,A -85,B 0,C 180,E1 -1188.9,E2 -1188.9} C_VEL
LIN {X 0,Y 594.893,Z 268.109,A -85,B 0,C 180,E1 -1191.847,E2 -1191.847} C_VEL
LIN {X 0,Y 595.091,Z 242.207,A -85,B 0,C 180,E1 -1194.802,E2 -1194.802} C_VEL
LIN {X 0,Y 594.997,Z 234.284,A -85,B 0,C 180,E1 -1195.726,E2 -1195.726} C_VEL
LIN {X 0,Y 594.349,Z 231.528,A -85,B 0,C 180,E1 -1196.109,E2 -1196.109} C_VEL
LIN {X 0,Y 594.327,Z 231.451,A -85,B 0,C 180,E1 -1199,E2 -1199} C_VEL
LIN {X 0,Y 594.349,Z 231.452,A -85,B 0,C 180,E1 -1201.638,E2 -1201.638} C_VEL
LIN {X 0,Y 594.343,Z 231.446,A -85,B 0,C 180,E1 -1204.581,E2 -1204.581} C_VEL
LIN {X 0,Y 594.346,Z 231.451,A -85,B 0,C 180,E1 -1207.603,E2 -1207.603} C_VEL
LIN {X 0,Y 594.33,Z 231.447,A -85,B 0,C 180,E1 -1210.569,E2 -1210.569} C_VEL
LIN {X 0,Y 594.332,Z 231.457,A -85,B 0,C 180,E1 -1213.301,E2 -1213.301} C_VEL
LIN {X 0,Y 594.329,Z 231.447,A -85,B 0,C 180,E1 -1216.163,E2 -1216.163} C_VEL
LIN {X 0,Y 594.351,Z 231.455,A -85,B 0,C 180,E1 -1219.179,E2 -1219.179} C_VEL
LIN {X 0,Y 594.339,Z 231.446,A -85,B 0,C 180,E1 -1222.056,E2 -1222.056} C_VEL
LIN {X 0,Y 594.311,Z 231.453,A -85,B 0,C 180,E1 -1224.68,E2 -1224.68} C_VEL
LIN {X 0,Y 594.325,Z 231.457,A -85,B 0,C 180,E1 -1227.094,E2 -1227.094} C_VEL
LIN {X 0,Y 594.333,Z 231.447,A -85,B 0,C 180,E1 -1229.678,E2 -1229.678} C_VEL
LIN {X 0,Y 594.307,Z 231.45,A -85,B 0,C 180,E1 -1231.769,E2 -1231.769} C_VEL
LIN {X 0,Y 594.324,Z 231.447,A -85,B 0,C 180,E1 -1234.053,E2 -1234.053} C_VEL
LIN {X 0,Y 594.33,Z 231.455,A -85,B 0,C 180,E1 -1237.031,E2 -1237.031} C_VEL
LIN {X 0,Y 594.333,Z 231.446,A -85,B 0,C 180,E1 -1239.945,E2 -1239.945} C_VEL
LIN {X 0,Y 594.353,Z 231.454,A -85,B 0,C 180,E1 -1242.806,E2 -1242.806} C_VEL
LIN {X 0,Y 594.314,Z 231.449,A -85,B 0,C 180,E1 -1245.849,E2 -1245.849} C_VEL
LIN {X 0,Y 594.353,Z 231.45,A -85,B 0,C 180,E1 -1248.937,E2 -1248.937} C_VEL
LIN {X 0,Y 594.325,Z 231.448,A -85,B 0,C 180,E1 -1251.842,E2 -1251.842} C_VEL
LIN {X 0,Y 594.369,Z 231.452,A -85,B 0,C 180,E1 -1254.572,E2 -1254.572} C_VEL
LIN {X 0,Y 594.354,Z 231.444,A -85,B 0,C 180,E1 -1257.289,E2 -1257.289} C_VEL
LIN {X 0,Y 594.37,Z 231.444,A -85,B 0,C 180,E1 -1260,E2 -1260} C_VEL
LIN {X 0,Y 594.386,Z 231.446,A -85,B 0,C 180,E1 -1262.711,E2 -1262.711} C_VEL
LIN {X 0,Y 594.334,Z 231.446,A -85,B 0,C 180,E1 -1265.428,E2 -1265.428} C_VEL
LIN {X 0,Y 594.336,Z 231.453,A -85,B 0,C 180,E1 -1268.158,E2 -1268.158} C_VEL
LIN {X 0,Y 594.315,Z 231.449,A -85,B 0,C 180,E1 -1271.044,E2 -1271.044} C_VEL
LIN {X 0,Y 594.331,Z 231.448,A -85,B 0,C 180,E1 -1273.68,E2 -1273.68} C_VEL
LIN {X 0,Y 594.312,Z 231.449,A -85,B 0,C 180,E1 -1275.325,E2 -1275.325} C_VEL
LIN {X 0,Y 593.64,Z 231.538,A -85,B 0,C 180,E1 -1275.891,E2 -1275.891} C_VEL
LIN {X 0,Y 590.775,Z 231.9,A -85,B 0,C 180,E1 -1276.809,E2 -1276.809} C_VEL
LIN {X 0,Y 588.364,Z 232.202,A -85,B 0,C 180,E1 -1277.547,E2 -1277.547} C_VEL
LIN {X 0,Y 587.343,Z 232.326,A -85,B 0,C 180,E1 -1278.117,E2 -1278.117} C_VEL
LIN {X 0,Y 587.268,Z 232.333,A -85,B 0,C 180,E1 -1278.31,E2 -1278.31} C_VEL
LIN {X 0,Y 587.301,Z 232.322,A -85,B 0,C 180,E1 -1281.039,E2 -1281.039} C_VEL
LIN {X 0,Y 587.303,Z 232.331,A -85,B 0,C 180,E1 -1284.008,E2 -1284.008} C_VEL
LIN {X 0,Y 587.276,Z 232.325,A -85,B 0,C 180,E1 -1287.049,E2 -1287.049} C_VEL
LIN {X 0,Y 587.301,Z 232.33,A -85,B 0,C 180,E1 -1290.172,E2 -1290.172} C_VEL
LIN {X 0,Y 587.297,Z 232.324,A -85,B 0,C 180,E1 -1292.582,E2 -1292.582} C_VEL
LIN {X 0,Y 587.278,Z 232.325,A -85,B 0,C 180,E1 -1295.059,E2 -1295.059} C_VEL
LIN {X 0,Y 587.294,Z 232.333,A -85,B 0,C 180,E1 -1297.835,E2 -1297.835} C_VEL
LIN {X 0,Y 587.276,Z 232.329,A -85,B 0,C 180,E1 -1300.258,E2 -1300.258} C_VEL
LIN {X 0,Y 587.268,Z 232.327,A -85,B 0,C 180,E1 -1303.115,E2 -1303.115} C_VEL
LIN {X 0,Y 587.29,Z 232.329,A -85,B 0,C 180,E1 -1306.048,E2 -1306.048} C_VEL
LIN {X 0,Y 587.273,Z 232.326,A -85,B 0,C 180,E1 -1308.933,E2 -1308.933} C_VEL
LIN {X 0,Y 587.299,Z 232.33,A -85,B 0,C 180,E1 -1311.52,E2 -1311.52} C_VEL
LIN {X 0,Y 587.265,Z 232.33,A -85,B 0,C 180,E1 -1314.099,E2 -1314.099} C_VEL
LIN {X 0,Y 587.301,Z 232.323,A -85,B 0,C 180,E1 -1316.895,E2 -1316.895} C_VEL
LIN {X 0,Y 587.288,Z 232.329,A -85,B 0,C 180,E1 -1319.828,E2 -1319.828} C_VEL
LIN {X 0,Y 587.286,Z 232.324,A -85,B 0,C 180,E1 -1322.32,E2 -1322.32} C_VEL
LIN {X 0,Y 587.283,Z 232.332,A -85,B 0,C 180,E1 -1325.239,E2 -1325.239} C_VEL
LIN {X 0,Y 587.294,Z 232.332,A -85,B 0,C 180,E1 -1327.485,E2 -1327.485} C_VEL
LIN {X 0,Y 587.306,Z 232.326,A -85,B 0,C 180,E1 -1329.695,E2 -1329.695} C_VEL
LIN {X 0,Y 587.27,Z 232.328,A -85,B 0,C 180,E1 -1331.872,E2 -1331.872} C_VEL
LIN {X 0,Y 587.283,Z 232.325,A -85,B 0,C 180,E1 -1334.024,E2 -1334.024} C_VEL
LIN {X 0,Y 587.311,Z 232.321,A -85,B 0,C 180,E1 -1336.154,E2 -1336.154} C_VEL
LIN {X 0,Y 587.342,Z 232.324,A -85,B 0,C 180,E1 -1338.963,E2 -1338.963} C_VEL
LIN {X 0,Y 587.287,Z 232.328,A -85,B 0,C 180,E1 -1341.744,E2 -1341.744} C_VEL
LIN {X 0,Y 587.32,Z 232.327,A -85,B 0,C 180,E1 -1344.507,E2 -1344.507} C_VEL
LIN {X 0,Y 587.374,Z 232.703,A -85,B 0,C 180,E1 -1344.68,E2 -1344.68} C_VEL
LIN {X 0,Y 587.77,Z 234.156,A -85,B 0,C 180,E1 -1344.769,E2 -1344.769} C_VEL
LIN {X 0,Y 587.74,Z 325.323,A -85,B 0,C 180,E1 -1345.908,E2 -1345.908} C_VEL
LIN {X 0,Y 587.685,Z 338.292,A -85,B 0,C 180,E1 -1346.208,E2 -1346.208} C_VEL
LIN {X 0,Y 587.616,Z 351.346,A -85,B 0,C 180,E1 -1346.658,E2 -1346.658} C_VEL
LIN {X 0,Y 587.526,Z 362.381,A -85,B 0,C 180,E1 -1347.172,E2 -1347.172} C_VEL
LIN {X 0,Y 587.434,Z 373.861,A -85,B 0,C 180,E1 -1347.858,E2 -1347.858} C_VEL
LIN {X 0,Y 587.392,Z 384.188,A -85,B 0,C 180,E1 -1348.629,E2 -1348.629} C_VEL
LIN {X 0,Y 587.318,Z 393.555,A -85,B 0,C 180,E1 -1349.486,E2 -1349.486} C_VEL
LIN {X 0,Y 587.258,Z 402.6,A -85,B 0,C 180,E1 -1350.515,E2 -1350.515} C_VEL
LIN {X 0,Y 587.209,Z 409.914,A -85,B 0,C 180,E1 -1351.543,E2 -1351.543} C_VEL
LIN {X 0,Y 587.162,Z 416.662,A -85,B 0,C 180,E1 -1352.744,E2 -1352.744} C_VEL
LIN {X 0,Y 587.213,Z 421.127,A -85,B 0,C 180,E1 -1353.774,E2 -1353.774} C_VEL
LIN {X 0,Y 587.131,Z 424.534,A -85,B 0,C 180,E1 -1354.807,E2 -1354.807} C_VEL
LIN {X 0,Y 587.18,Z 426.23,A -85,B 0,C 180,E1 -1355.495,E2 -1355.495} C_VEL
LIN {X 0,Y 587.167,Z 428.414,A -85,B 0,C 180,E1 -1356.875,E2 -1356.875} C_VEL
LIN {X 0,Y 587.146,Z 428.897,A -85,B 0,C 180,E1 -1357.566,E2 -1357.566} C_VEL
LIN {X 0,Y 587.127,Z 428.633,A -85,B 0,C 180,E1 -1358.952,E2 -1358.952} C_VEL
LIN {X 0,Y 587.151,Z 427.917,A -85,B 0,C 180,E1 -1359.647,E2 -1359.647} C_VEL
LIN {X 0,Y 587.141,Z 426.754,A -85,B 0,C 180,E1 -1360.343,E2 -1360.343} C_VEL
LIN {X 0,Y 587.15,Z 424.221,A -85,B 0,C 180,E1 -1361.391,E2 -1361.391} C_VEL
LIN {X 0,Y 587.182,Z 420.643,A -85,B 0,C 180,E1 -1362.441,E2 -1362.441} C_VEL
LIN {X 0,Y 587.197,Z 415.905,A -85,B 0,C 180,E1 -1363.497,E2 -1363.497} C_VEL
LIN {X 0,Y 587.221,Z 409.851,A -85,B 0,C 180,E1 -1364.556,E2 -1364.556} C_VEL
LIN {X 0,Y 587.26,Z 402.244,A -85,B 0,C 180,E1 -1365.621,E2 -1365.621} C_VEL
LIN {X 0,Y 587.298,Z 394.439,A -85,B 0,C 180,E1 -1366.511,E2 -1366.511} C_VEL
LIN {X 0,Y 587.407,Z 384.878,A -85,B 0,C 180,E1 -1367.404,E2 -1367.404} C_VEL
LIN {X 0,Y 587.45,Z 374.147,A -85,B 0,C 180,E1 -1368.213,E2 -1368.213} C_VEL
LIN {X 0,Y 587.556,Z 362.367,A -85,B 0,C 180,E1 -1368.918,E2 -1368.918} C_VEL
LIN {X 0,Y 587.608,Z 349.948,A -85,B 0,C 180,E1 -1369.487,E2 -1369.487} C_VEL
LIN {X 0,Y 587.684,Z 336.734,A -85,B 0,C 180,E1 -1369.927,E2 -1369.927} C_VEL
LIN {X 0,Y 587.774,Z 324.483,A -85,B 0,C 180,E1 -1370.197,E2 -1370.197} C_VEL
LIN {X 0,Y 587.743,Z 234.016,A -85,B 0,C 180,E1 -1371.324,E2 -1371.324} C_VEL
LIN {X 0,Y 587.385,Z 232.699,A -85,B 0,C 180,E1 -1371.41,E2 -1371.41} C_VEL
LIN {X 0,Y 587.331,Z 232.36,A -85,B 0,C 180,E1 -1371.503,E2 -1371.503} C_VEL
LIN {X 0,Y 587.315,Z 232.327,A -85,B 0,C 180,E1 -1374.571,E2 -1374.571} C_VEL
LIN {X 0,Y 587.304,Z 232.33,A -85,B 0,C 180,E1 -1377.047,E2 -1377.047} C_VEL
LIN {X 0,Y 587.312,Z 232.323,A -85,B 0,C 180,E1 -1379.381,E2 -1379.381} C_VEL
LIN {X 0,Y 587.341,Z 232.316,A -85,B 0,C 180,E1 -1381.834,E2 -1381.834} C_VEL
LIN {X 0,Y 587.336,Z 232.323,A -85,B 0,C 180,E1 -1384.345,E2 -1384.345} C_VEL
LIN {X 0,Y 587.308,Z 232.32,A -85,B 0,C 180,E1 -1387.61,E2 -1387.61} C_VEL
LIN {X 0,Y 587.301,Z 232.327,A -85,B 0,C 180,E1 -1390.255,E2 -1390.255} C_VEL
LIN {X 0,Y 587.301,Z 232.326,A -85,B 0,C 180,E1 -1393.007,E2 -1393.007} C_VEL
LIN {X 0,Y 587.297,Z 232.326,A -85,B 0,C 180,E1 -1396.046,E2 -1396.046} C_VEL
LIN {X 0,Y 587.325,Z 232.323,A -85,B 0,C 180,E1 -1398.925,E2 -1398.925} C_VEL
LIN {X 0,Y 587.306,Z 232.321,A -85,B 0,C 180,E1 -1401.518,E2 -1401.518} C_VEL
LIN {X 0,Y 587.275,Z 232.33,A -85,B 0,C 180,E1 -1404.098,E2 -1404.098} C_VEL
LIN {X 0,Y 587.323,Z 232.325,A -85,B 0,C 180,E1 -1406.602,E2 -1406.602} C_VEL
LIN {X 0,Y 587.322,Z 232.318,A -85,B 0,C 180,E1 -1409.491,E2 -1409.491} C_VEL
LIN {X 0,Y 587.293,Z 232.333,A -85,B 0,C 180,E1 -1412.179,E2 -1412.179} C_VEL
LIN {X 0,Y 587.339,Z 232.318,A -85,B 0,C 180,E1 -1415.241,E2 -1415.241} C_VEL
LIN {X 0,Y 587.299,Z 232.328,A -85,B 0,C 180,E1 -1418.225,E2 -1418.225} C_VEL
LIN {X 0,Y 587.322,Z 232.319,A -85,B 0,C 180,E1 -1421.15,E2 -1421.15} C_VEL
LIN {X 0,Y 587.294,Z 232.332,A -85,B 0,C 180,E1 -1424.024,E2 -1424.024} C_VEL
LIN {X 0,Y 587.339,Z 232.324,A -85,B 0,C 180,E1 -1426.154,E2 -1426.154} C_VEL
LIN {X 0,Y 587.328,Z 232.319,A -85,B 0,C 180,E1 -1428.962,E2 -1428.962} C_VEL
LIN {X 0,Y 587.326,Z 232.327,A -85,B 0,C 180,E1 -1431.744,E2 -1431.744} C_VEL
LIN {X 0,Y 587.317,Z 232.321,A -85,B 0,C 180,E1 -1434.506,E2 -1434.506} C_VEL
LIN {X 0,Y 587.353,Z 232.318,A -85,B 0,C 180,E1 -1437.256,E2 -1437.256} C_VEL
LIN {X 0,Y 587.358,Z 232.32,A -85,B 0,C 180,E1 -1440,E2 -1440} C_VEL
LIN {X 0,Y 587.332,Z 232.318,A -85,B 0,C 180,E1 -1442.743,E2 -1442.743} C_VEL
LIN {X 0,Y 587.338,Z 232.327,A -85,B 0,C 180,E1 -1445.493,E2 -1445.493} C_VEL
LIN {X 0,Y 587.305,Z 232.322,A -85,B 0,C 180,E1 -1448.256,E2 -1448.256} C_VEL
LIN {X 0,Y 587.34,Z 232.323,A -85,B 0,C 180,E1 -1451.134,E2 -1451.134} C_VEL
LIN {X 0,Y 587.292,Z 232.324,A -85,B 0,C 180,E1 -1454.236,E2 -1454.236} C_VEL
LIN {X 0,Y 587.313,Z 232.323,A -85,B 0,C 180,E1 -1456.805,E2 -1456.805} C_VEL
LIN {X 0,Y 587.29,Z 232.329,A -85,B 0,C 180,E1 -1459.577,E2 -1459.577} C_VEL
LIN {X 0,Y 587.293,Z 232.325,A -85,B 0,C 180,E1 -1461.775,E2 -1461.775} C_VEL
LIN {X 0,Y 587.288,Z 232.328,A -85,B 0,C 180,E1 -1464.761,E2 -1464.761} C_VEL
LIN {X 0,Y 587.288,Z 232.325,A -85,B 0,C 180,E1 -1467.683,E2 -1467.683} C_VEL
LIN {X 0,Y 587.284,Z 232.325,A -85,B 0,C 180,E1 -1470.173,E2 -1470.173} C_VEL
LIN {X 0,Y 587.321,Z 232.328,A -85,B 0,C 180,E1 -1473.11,E2 -1473.11} C_VEL
LIN {X 0,Y 587.259,Z 232.33,A -85,B 0,C 180,E1 -1475.534,E2 -1475.534} C_VEL
LIN {X 0,Y 587.301,Z 232.322,A -85,B 0,C 180,E1 -1477.835,E2 -1477.835} C_VEL
LIN {X 0,Y 587.292,Z 232.325,A -85,B 0,C 180,E1 -1480.256,E2 -1480.256} C_VEL
LIN {X 0,Y 587.281,Z 232.33,A -85,B 0,C 180,E1 -1483.116,E2 -1483.116} C_VEL
LIN {X 0,Y 587.281,Z 232.326,A -85,B 0,C 180,E1 -1486.046,E2 -1486.046} C_VEL
LIN {X 0,Y 587.303,Z 232.328,A -85,B 0,C 180,E1 -1488.929,E2 -1488.929} C_VEL
LIN {X 0,Y 587.265,Z 232.327,A -85,B 0,C 180,E1 -1491.516,E2 -1491.516} C_VEL
LIN {X 0,Y 587.257,Z 232.331,A -85,B 0,C 180,E1 -1494.098,E2 -1494.098} C_VEL
LIN {X 0,Y 587.308,Z 232.332,A -85,B 0,C 180,E1 -1496.602,E2 -1496.602} C_VEL
LIN {X 0,Y 587.282,Z 232.326,A -85,B 0,C 180,E1 -1499.5,E2 -1499.5} C_VEL
LIN {X 0,Y 587.292,Z 232.333,A -85,B 0,C 180,E1 -1502.319,E2 -1502.319} C_VEL
LIN {X 0,Y 587.333,Z 232.505,A -85,B 0,C 180,E1 -1503.789,E2 -1503.789} C_VEL
LIN {X 0,Y 588.213,Z 236.996,A -85,B 0,C 180,E1 -1504.335,E2 -1504.335} C_VEL
LIN {X 0,Y 588.175,Z 251.997,A -85,B 0,C 180,E1 -1506.03,E2 -1506.03} C_VEL
LIN {X 0,Y 587.997,Z 276.078,A -85,B 0,C 180,E1 -1508.795,E2 -1508.795} C_VEL
LIN {X 0,Y 587.764,Z 301.928,A -85,B 0,C 180,E1 -1511.707,E2 -1511.707} C_VEL
LIN {X 0,Y 587.575,Z 326.088,A -85,B 0,C 180,E1 -1514.388,E2 -1514.388} C_VEL
LIN {X 0,Y 587.5,Z 345.146,A -85,B 0,C 180,E1 -1516.466,E2 -1516.466} C_VEL
LIN {X 0,Y 587.873,Z 348.932,A -85,B 0,C 180,E1 -1516.541,E2 -1516.541} C_VEL
LIN {X 0,Y 587.721,Z 454.946,A -85,B 0,C 180,E1 -1517.855,E2 -1517.855} C_VEL
LIN {X 0,Y 587.681,Z 468.218,A -85,B 0,C 180,E1 -1518.161,E2 -1518.161} C_VEL
LIN {X 0,Y 587.627,Z 480.754,A -85,B 0,C 180,E1 -1518.59,E2 -1518.59} C_VEL
LIN {X 0,Y 587.554,Z 492.63,A -85,B 0,C 180,E1 -1519.141,E2 -1519.141} C_VEL
LIN {X 0,Y 587.467,Z 504.201,A -85,B 0,C 180,E1 -1519.836,E2 -1519.836} C_VEL
LIN {X 0,Y 587.392,Z 514.597,A -85,B 0,C 180,E1 -1520.618,E2 -1520.618} C_VEL
LIN {X 0,Y 587.322,Z 523.111,A -85,B 0,C 180,E1 -1521.397,E2 -1521.397} C_VEL
LIN {X 0,Y 587.274,Z 530.96,A -85,B 0,C 180,E1 -1522.263,E2 -1522.263} C_VEL
LIN {X 0,Y 587.23,Z 537.468,A -85,B 0,C 180,E1 -1523.126,E2 -1523.126} C_VEL
LIN {X 0,Y 587.236,Z 543.866,A -85,B 0,C 180,E1 -1524.161,E2 -1524.161} C_VEL
LIN {X 0,Y 587.147,Z 548.949,A -85,B 0,C 180,E1 -1525.193,E2 -1525.193} C_VEL
LIN {X 0,Y 587.212,Z 552.895,A -85,B 0,C 180,E1 -1526.226,E2 -1526.226} C_VEL
LIN {X 0,Y 587.132,Z 555.808,A -85,B 0,C 180,E1 -1527.255,E2 -1527.255} C_VEL
LIN {X 0,Y 587.141,Z 557.2,A -85,B 0,C 180,E1 -1527.942,E2 -1527.942} C_VEL
LIN {X 0,Y 587.14,Z 558.784,A -85,B 0,C 180,E1 -1529.314,E2 -1529.314} C_VEL
LIN {X 0,Y 587.137,Z 559,A -85,B 0,C 180,E1 -1530,E2 -1530} C_VEL
LIN {X 0,Y 587.147,Z 558.186,A -85,B 0,C 180,E1 -1531.371,E2 -1531.371} C_VEL
LIN {X 0,Y 587.141,Z 557.201,A -85,B 0,C 180,E1 -1532.058,E2 -1532.058} C_VEL
LIN {X 0,Y 587.132,Z 555.81,A -85,B 0,C 180,E1 -1532.744,E2 -1532.744} C_VEL
LIN {X 0,Y 587.212,Z 552.897,A -85,B 0,C 180,E1 -1533.774,E2 -1533.774} C_VEL
LIN {X 0,Y 587.147,Z 548.951,A -85,B 0,C 180,E1 -1534.806,E2 -1534.806} C_VEL
LIN {X 0,Y 587.217,Z 542.88,A -85,B 0,C 180,E1 -1536.011,E2 -1536.011} C_VEL
LIN {X 0,Y 587.244,Z 536.24,A -85,B 0,C 180,E1 -1537.046,E2 -1537.046} C_VEL
LIN {X 0,Y 587.299,Z 527.994,A -85,B 0,C 180,E1 -1538.083,E2 -1538.083} C_VEL
LIN {X 0,Y 587.343,Z 519.543,A -85,B 0,C 180,E1 -1538.948,E2 -1538.948} C_VEL
LIN {X 0,Y 587.418,Z 509.103,A -85,B 0,C 180,E1 -1539.816,E2 -1539.816} C_VEL
LIN {X 0,Y 587.489,Z 498.766,A -85,B 0,C 180,E1 -1540.511,E2 -1540.511} C_VEL
LIN {X 0,Y 587.583,Z 486.809,A -85,B 0,C 180,E1 -1541.149,E2 -1541.149} C_VEL
LIN {X 0,Y 587.631,Z 474.605,A -85,B 0,C 180,E1 -1541.639,E2 -1541.639} C_VEL
LIN {X 0,Y 587.725,Z 461.459,A -85,B 0,C 180,E1 -1542.013,E2 -1542.013} C_VEL
LIN {X 0,Y 587.762,Z 449.126,A -85,B 0,C 180,E1 -1542.231,E2 -1542.231} C_VEL
LIN {X 0,Y 587.774,Z 347.191,A -85,B 0,C 180,E1 -1543.483,E2 -1543.483} C_VEL
LIN {X 0,Y 587.499,Z 345.151,A -85,B 0,C 180,E1 -1543.533,E2 -1543.533} C_VEL
LIN {X 0,Y 587.642,Z 321.262,A -85,B 0,C 180,E1 -1546.144,E2 -1546.144} C_VEL
LIN {X 0,Y 587.826,Z 295.211,A -85,B 0,C 180,E1 -1549.045,E2 -1549.045} C_VEL
LIN {X 0,Y 588.026,Z 269.72,A -85,B 0,C 180,E1 -1551.931,E2 -1551.931} C_VEL
LIN {X 0,Y 588.264,Z 244.018,A -85,B 0,C 180,E1 -1554.886,E2 -1554.886} C_VEL
LIN {X 0,Y 588.242,Z 237.026,A -85,B 0,C 180,E1 -1555.663,E2 -1555.663} C_VEL
LIN {X 0,Y 587.323,Z 232.443,A -85,B 0,C 180,E1 -1556.233,E2 -1556.233} C_VEL
LIN {X 0,Y 587.29,Z 232.329,A -85,B 0,C 180,E1 -1559.122,E2 -1559.122} C_VEL
LIN {X 0,Y 587.31,Z 232.326,A -85,B 0,C 180,E1 -1561.83,E2 -1561.83} C_VEL
LIN {X 0,Y 587.314,Z 232.321,A -85,B 0,C 180,E1 -1564.343,E2 -1564.343} C_VEL
LIN {X 0,Y 587.299,Z 232.329,A -85,B 0,C 180,E1 -1567.61,E2 -1567.61} C_VEL
LIN {X 0,Y 587.279,Z 232.325,A -85,B 0,C 180,E1 -1570.256,E2 -1570.256} C_VEL
LIN {X 0,Y 587.274,Z 232.333,A -85,B 0,C 180,E1 -1573.114,E2 -1573.114} C_VEL
LIN {X 0,Y 587.286,Z 232.325,A -85,B 0,C 180,E1 -1576.046,E2 -1576.046} C_VEL
LIN {X 0,Y 587.29,Z 232.33,A -85,B 0,C 180,E1 -1578.928,E2 -1578.928} C_VEL
LIN {X 0,Y 587.296,Z 232.327,A -85,B 0,C 180,E1 -1581.518,E2 -1581.518} C_VEL
LIN {X 0,Y 587.255,Z 232.328,A -85,B 0,C 180,E1 -1584.097,E2 -1584.097} C_VEL
LIN {X 0,Y 587.29,Z 232.327,A -85,B 0,C 180,E1 -1586.6,E2 -1586.6} C_VEL
LIN {X 0,Y 587.292,Z 232.326,A -85,B 0,C 180,E1 -1589.495,E2 -1589.495} C_VEL
LIN {X 0,Y 587.282,Z 232.326,A -85,B 0,C 180,E1 -1592.317,E2 -1592.317} C_VEL
LIN {X 0,Y 587.28,Z 232.33,A -85,B 0,C 180,E1 -1595.238,E2 -1595.238} C_VEL
LIN {X 0,Y 587.283,Z 232.326,A -85,B 0,C 180,E1 -1598.224,E2 -1598.224} C_VEL
LIN {X 0,Y 587.31,Z 232.326,A -85,B 0,C 180,E1 -1601.15,E2 -1601.15} C_VEL
LIN {X 0,Y 587.275,Z 232.326,A -85,B 0,C 180,E1 -1604.024,E2 -1604.024} C_VEL
LIN {X 0,Y 587.27,Z 232.334,A -85,B 0,C 180,E1 -1606.857,E2 -1606.857} C_VEL
LIN {X 0,Y 587.322,Z 232.325,A -85,B 0,C 180,E1 -1608.962,E2 -1608.962} C_VEL
LIN {X 0,Y 587.293,Z 232.323,A -85,B 0,C 180,E1 -1611.744,E2 -1611.744} C_VEL
LIN {X 0,Y 587.331,Z 232.327,A -85,B 0,C 180,E1 -1614.507,E2 -1614.507} C_VEL
LIN {X 0,Y 587.325,Z 232.32,A -85,B 0,C 180,E1 -1617.257,E2 -1617.257} C_VEL
LIN {X 0,Y 587.341,Z 232.32,A -85,B 0,C 180,E1 -1620,E2 -1620} C_VEL
LIN {X 0,Y 587.348,Z 232.322,A -85,B 0,C 180,E1 -1622.744,E2 -1622.744} C_VEL
LIN {X 0,Y 587.303,Z 232.322,A -85,B 0,C 180,E1 -1625.494,E2 -1625.494} C_VEL
LIN {X 0,Y 587.302,Z 232.331,A -85,B 0,C 180,E1 -1628.256,E2 -1628.256} C_VEL
LIN {X 0,Y 587.281,Z 232.325,A -85,B 0,C 180,E1 -1631.108,E2 -1631.108} C_VEL
LIN {X 0,Y 587.318,Z 232.324,A -85,B 0,C 180,E1 -1633.847,E2 -1633.847} C_VEL
LIN {X 0,Y 587.283,Z 232.327,A -85,B 0,C 180,E1 -1636.798,E2 -1636.798} C_VEL
LIN {X 0,Y 587.268,Z 232.333,A -85,B 0,C 180,E1 -1638.31,E2 -1638.31} C_VEL
LIN {X 0,Y 586.631,Z 232.408,A -85,B 0,C 180,E1 -1638.882,E2 -1638.882} C_VEL
LIN {X 0,Y 583.819,Z 232.76,A -85,B 0,C 180,E1 -1639.811,E2 -1639.811} C_VEL
LIN {X 0,Y 581.414,Z 233.06,A -85,B 0,C 180,E1 -1640.558,E2 -1640.558} C_VEL
LIN {X 0,Y 580.357,Z 233.188,A -85,B 0,C 180,E1 -1641.134,E2 -1641.134} C_VEL
LIN {X 0,Y 580.259,Z 233.2,A -85,B 0,C 180,E1 -1641.33,E2 -1641.33} C_VEL
LIN {X 0,Y 580.25,Z 233.203,A -85,B 0,C 180,E1 -1643.56,E2 -1643.56} C_VEL
LIN {X 0,Y 580.24,Z 233.208,A -85,B 0,C 180,E1 -1646.327,E2 -1646.327} C_VEL
LIN {X 0,Y 580.24,Z 233.203,A -85,B 0,C 180,E1 -1649.302,E2 -1649.302} C_VEL
LIN {X 0,Y 580.266,Z 233.205,A -85,B 0,C 180,E1 -1652.203,E2 -1652.203} C_VEL
LIN {X 0,Y 580.258,Z 233.2,A -85,B 0,C 180,E1 -1654.699,E2 -1654.699} C_VEL
LIN {X 0,Y 580.253,Z 233.202,A -85,B 0,C 180,E1 -1657.272,E2 -1657.272} C_VEL
LIN {X 0,Y 580.238,Z 233.206,A -85,B 0,C 180,E1 -1660.266,E2 -1660.266} C_VEL
LIN {X 0,Y 580.233,Z 233.203,A -85,B 0,C 180,E1 -1662.711,E2 -1662.711} C_VEL
LIN {X 0,Y 580.24,Z 233.21,A -85,B 0,C 180,E1 -1665.613,E2 -1665.613} C_VEL
LIN {X 0,Y 580.23,Z 233.206,A -85,B 0,C 180,E1 -1668.228,E2 -1668.228} C_VEL
LIN {X 0,Y 580.25,Z 233.202,A -85,B 0,C 180,E1 -1670.964,E2 -1670.964} C_VEL
LIN {X 0,Y 580.231,Z 233.213,A -85,B 0,C 180,E1 -1673.595,E2 -1673.595} C_VEL
LIN {X 0,Y 580.251,Z 233.203,A -85,B 0,C 180,E1 -1676.142,E2 -1676.142} C_VEL
LIN {X 0,Y 580.226,Z 233.204,A -85,B 0,C 180,E1 -1678.613,E2 -1678.613} C_VEL
LIN {X 0,Y 580.264,Z 233.202,A -85,B 0,C 180,E1 -1681.023,E2 -1681.023} C_VEL
LIN {X 0,Y 580.245,Z 233.208,A -85,B 0,C 180,E1 -1683.677,E2 -1683.677} C_VEL
LIN {X 0,Y 580.245,Z 233.201,A -85,B 0,C 180,E1 -1686.441,E2 -1686.441} C_VEL
LIN {X 0,Y 580.255,Z 233.209,A -85,B 0,C 180,E1 -1689.437,E2 -1689.437} C_VEL
LIN {X 0,Y 580.231,Z 233.208,A -85,B 0,C 180,E1 -1691.645,E2 -1691.645} C_VEL
LIN {X 0,Y 580.241,Z 233.204,A -85,B 0,C 180,E1 -1693.825,E2 -1693.825} C_VEL
LIN {X 0,Y 580.274,Z 233.198,A -85,B 0,C 180,E1 -1695.982,E2 -1695.982} C_VEL
LIN {X 0,Y 580.311,Z 233.198,A -85,B 0,C 180,E1 -1698.828,E2 -1698.828} C_VEL
LIN {X 0,Y 580.252,Z 233.206,A -85,B 0,C 180,E1 -1701.643,E2 -1701.643} C_VEL
LIN {X 0,Y 580.308,Z 233.29,A -85,B 0,C 180,E1 -1704.462,E2 -1704.462} C_VEL
LIN {X 0,Y 580.529,Z 234.372,A -85,B 0,C 180,E1 -1704.595,E2 -1704.595} C_VEL
LIN {X 0,Y 580.982,Z 236.548,A -85,B 0,C 180,E1 -1704.643,E2 -1704.643} C_VEL
LIN {X 0,Y 580.8,Z 324.789,A -85,B 0,C 180,E1 -1705.75,E2 -1705.75} C_VEL
LIN {X 0,Y 580.733,Z 337.938,A -85,B 0,C 180,E1 -1706.054,E2 -1706.054} C_VEL
LIN {X 0,Y 580.66,Z 350.535,A -85,B 0,C 180,E1 -1706.487,E2 -1706.487} C_VEL
LIN {X 0,Y 580.539,Z 362.589,A -85,B 0,C 180,E1 -1707.051,E2 -1707.051} C_VEL
LIN {X 0,Y 580.435,Z 374.028,A -85,B 0,C 180,E1 -1707.745,E2 -1707.745} C_VEL
LIN {X 0,Y 580.353,Z 384.333,A -85,B 0,C 180,E1 -1708.526,E2 -1708.526} C_VEL
LIN {X 0,Y 580.273,Z 392.801,A -85,B 0,C 180,E1 -1709.306,E2 -1709.306} C_VEL
LIN {X 0,Y 580.221,Z 400.63,A -85,B 0,C 180,E1 -1710.174,E2 -1710.174} C_VEL
LIN {X 0,Y 580.171,Z 408.318,A -85,B 0,C 180,E1 -1711.215,E2 -1711.215} C_VEL
LIN {X 0,Y 580.112,Z 415.406,A -85,B 0,C 180,E1 -1712.43,E2 -1712.43} C_VEL
LIN {X 0,Y 580.127,Z 420.145,A -85,B 0,C 180,E1 -1713.473,E2 -1713.473} C_VEL
LIN {X 0,Y 580.104,Z 423.79,A -85,B 0,C 180,E1 -1714.517,E2 -1714.517} C_VEL
LIN {X 0,Y 580.099,Z 426.435,A -85,B 0,C 180,E1 -1715.562,E2 -1715.562} C_VEL
LIN {X 0,Y 580.101,Z 428.078,A -85,B 0,C 180,E1 -1716.562,E2 -1716.562} C_VEL
LIN {X 0,Y 580.067,Z 428.919,A -85,B 0,C 180,E1 -1717.659,E2 -1717.659} C_VEL
LIN {X 0,Y 580.061,Z 428.935,A -85,B 0,C 180,E1 -1718.36,E2 -1718.36} C_VEL
LIN {X 0,Y 580.026,Z 428.563,A -85,B 0,C 180,E1 -1719.063,E2 -1719.063} C_VEL
LIN {X 0,Y 580.058,Z 427.775,A -85,B 0,C 180,E1 -1719.766,E2 -1719.766} C_VEL
LIN {X 0,Y 580.075,Z 425.171,A -85,B 0,C 180,E1 -1721.075,E2 -1721.075} C_VEL
LIN {X 0,Y 580.081,Z 421.581,A -85,B 0,C 180,E1 -1722.241,E2 -1722.241} C_VEL
LIN {X 0,Y 580.097,Z 417.135,A -85,B 0,C 180,E1 -1723.308,E2 -1723.308} C_VEL
LIN {X 0,Y 580.153,Z 411.017,A -85,B 0,C 180,E1 -1724.451,E2 -1724.451} C_VEL
LIN {X 0,Y 580.199,Z 404.245,A -85,B 0,C 180,E1 -1725.455,E2 -1725.455} C_VEL
LIN {X 0,Y 580.248,Z 395.165,A -85,B 0,C 180,E1 -1726.537,E2 -1726.537} C_VEL
LIN {X 0,Y 580.359,Z 385.801,A -85,B 0,C 180,E1 -1727.44,E2 -1727.44} C_VEL
LIN {X 0,Y 580.448,Z 375.297,A -85,B 0,C 180,E1 -1728.258,E2 -1728.258} C_VEL
LIN {X 0,Y 580.564,Z 363.535,A -85,B 0,C 180,E1 -1728.986,E2 -1728.986} C_VEL
LIN {X 0,Y 580.637,Z 351.748,A -85,B 0,C 180,E1 -1729.555,E2 -1729.555} C_VEL
LIN {X 0,Y 580.722,Z 338.692,A -85,B 0,C 180,E1 -1730.015,E2 -1730.015} C_VEL
LIN {X 0,Y 580.821,Z 325.064,A -85,B 0,C 180,E1 -1730.334,E2 -1730.334} C_VEL
LIN {X 0,Y 580.811,Z 235.3,A -85,B 0,C 180,E1 -1731.467,E2 -1731.467} C_VEL
LIN {X 0,Y 580.401,Z 233.781,A -85,B 0,C 180,E1 -1731.539,E2 -1731.539} C_VEL
LIN {X 0,Y 580.282,Z 233.227,A -85,B 0,C 180,E1 -1731.678,E2 -1731.678} C_VEL
LIN {X 0,Y 580.266,Z 233.203,A -85,B 0,C 180,E1 -1734.318,E2 -1734.318} C_VEL
LIN {X 0,Y 580.24,Z 233.21,A -85,B 0,C 180,E1 -1736.625,E2 -1736.625} C_VEL
LIN {X 0,Y 580.276,Z 233.201,A -85,B 0,C 180,E1 -1739.304,E2 -1739.304} C_VEL
LIN {X 0,Y 580.297,Z 233.195,A -85,B 0,C 180,E1 -1742.2,E2 -1742.2} C_VEL
LIN {X 0,Y 580.28,Z 233.206,A -85,B 0,C 180,E1 -1744.696,E2 -1744.696} C_VEL
LIN {X 0,Y 580.268,Z 233.198,A -85,B 0,C 180,E1 -1747.27,E2 -1747.27} C_VEL
LIN {X 0,Y 580.281,Z 233.202,A -85,B 0,C 180,E1 -1750.269,E2 -1750.269} C_VEL
LIN {X 0,Y 580.269,Z 233.207,A -85,B 0,C 180,E1 -1752.706,E2 -1752.706} C_VEL
LIN {X 0,Y 580.248,Z 233.201,A -85,B 0,C 180,E1 -1755.61,E2 -1755.61} C_VEL
LIN {X 0,Y 580.266,Z 233.206,A -85,B 0,C 180,E1 -1758.67,E2 -1758.67} C_VEL
LIN {X 0,Y 580.259,Z 233.201,A -85,B 0,C 180,E1 -1760.963,E2 -1760.963} C_VEL
LIN {X 0,Y 580.235,Z 233.202,A -85,B 0,C 180,E1 -1763.593,E2 -1763.593} C_VEL
LIN {X 0,Y 580.302,Z 233.202,A -85,B 0,C 180,E1 -1766.144,E2 -1766.144} C_VEL
LIN {X 0,Y 580.261,Z 233.201,A -85,B 0,C 180,E1 -1768.613,E2 -1768.613} C_VEL
LIN {X 0,Y 580.277,Z 233.197,A -85,B 0,C 180,E1 -1771.023,E2 -1771.023} C_VEL
LIN {X 0,Y 580.253,Z 233.211,A -85,B 0,C 180,E1 -1774.149,E2 -1774.149} C_VEL
LIN {X 0,Y 580.263,Z 233.201,A -85,B 0,C 180,E1 -1776.441,E2 -1776.441} C_VEL
LIN {X 0,Y 580.257,Z 233.198,A -85,B 0,C 180,E1 -1779.436,E2 -1779.436} C_VEL
LIN {X 0,Y 580.241,Z 233.205,A -85,B 0,C 180,E1 -1781.644,E2 -1781.644} C_VEL
LIN {X 0,Y 580.244,Z 233.209,A -85,B 0,C 180,E1 -1783.824,E2 -1783.824} C_VEL
LIN {X 0,Y 580.301,Z 233.204,A -85,B 0,C 180,E1 -1785.982,E2 -1785.982} C_VEL
LIN {X 0,Y 580.297,Z 233.195,A -85,B 0,C 180,E1 -1788.827,E2 -1788.827} C_VEL
LIN {X 0,Y 580.294,Z 233.201,A -85,B 0,C 180,E1 -1791.643,E2 -1791.643} C_VEL
LIN {X 0,Y 580.286,Z 233.197,A -85,B 0,C 180,E1 -1794.44,E2 -1794.44} C_VEL
LIN {X 0,Y 580.317,Z 233.194,A -85,B 0,C 180,E1 -1797.223,E2 -1797.223} C_VEL
LIN {X 0,Y 580.328,Z 233.195,A -85,B 0,C 180,E1 -1800,E2 -1800} C_VEL
LIN {X 0,Y 580.302,Z 233.194,A -85,B 0,C 180,E1 -1802.777,E2 -1802.777} C_VEL
LIN {X 0,Y 580.302,Z 233.204,A -85,B 0,C 180,E1 -1805.56,E2 -1805.56} C_VEL
LIN {X 0,Y 580.278,Z 233.197,A -85,B 0,C 180,E1 -1808.357,E2 -1808.357} C_VEL
LIN {X 0,Y 580.292,Z 233.201,A -85,B 0,C 180,E1 -1811.191,E2 -1811.191} C_VEL
LIN {X 0,Y 580.258,Z 233.199,A -85,B 0,C 180,E1 -1814.32,E2 -1814.32} C_VEL
LIN {X 0,Y 580.281,Z 233.2,A -85,B 0,C 180,E1 -1816.906,E2 -1816.906} C_VEL
LIN {X 0,Y 580.264,Z 233.202,A -85,B 0,C 180,E1 -1819.824,E2 -1819.824} C_VEL
LIN {X 0,Y 580.237,Z 233.202,A -85,B 0,C 180,E1 -1822.054,E2 -1822.054} C_VEL
LIN {X 0,Y 580.264,Z 233.208,A -85,B 0,C 180,E1 -1825.082,E2 -1825.082} C_VEL
LIN {X 0,Y 580.234,Z 233.202,A -85,B 0,C 180,E1 -1827.848,E2 -1827.848} C_VEL
LIN {X 0,Y 580.248,Z 233.205,A -85,B 0,C 180,E1 -1830.69,E2 -1830.69} C_VEL
LIN {X 0,Y 580.267,Z 233.202,A -85,B 0,C 180,E1 -1833.312,E2 -1833.312} C_VEL
LIN {X 0,Y 580.212,Z 233.206,A -85,B 0,C 180,E1 -1835.753,E2 -1835.753} C_VEL
LIN {X 0,Y 580.267,Z 233.199,A -85,B 0,C 180,E1 -1838.148,E2 -1838.148} C_VEL
LIN {X 0,Y 580.267,Z 233.208,A -85,B 0,C 180,E1 -1840.846,E2 -1840.846} C_VEL
LIN {X 0,Y 580.228,Z 233.204,A -85,B 0,C 180,E1 -1843.663,E2 -1843.663} C_VEL
LIN {X 0,Y 580.221,Z 233.212,A -85,B 0,C 180,E1 -1846.615,E2 -1846.615} C_VEL
LIN {X 0,Y 580.249,Z 233.203,A -85,B 0,C 180,E1 -1849.153,E2 -1849.153} C_VEL
LIN {X 0,Y 580.233,Z 233.203,A -85,B 0,C 180,E1 -1851.935,E2 -1851.935} C_VEL
LIN {X 0,Y 580.209,Z 233.214,A -85,B 0,C 180,E1 -1854.45,E2 -1854.45} C_VEL
LIN {X 0,Y 580.24,Z 233.206,A -85,B 0,C 180,E1 -1856.972,E2 -1856.972} C_VEL
LIN {X 0,Y 580.247,Z 233.203,A -85,B 0,C 180,E1 -1859.423,E2 -1859.423} C_VEL
LIN {X 0,Y 580.233,Z 233.21,A -85,B 0,C 180,E1 -1862.154,E2 -1862.154} C_VEL
LIN {X 0,Y 580.278,Z 233.353,A -85,B 0,C 180,E1 -1863.643,E2 -1863.643} C_VEL
LIN {X 0,Y 581.341,Z 239.513,A -85,B 0,C 180,E1 -1864.394,E2 -1864.394} C_VEL
LIN {X 0,Y 581.255,Z 264.882,A -85,B 0,C 180,E1 -1867.238,E2 -1867.238} C_VEL
LIN {X 0,Y 580.998,Z 289.043,A -85,B 0,C 180,E1 -1870.018,E2 -1870.018} C_VEL
LIN {X 0,Y 580.732,Z 316.424,A -85,B 0,C 180,E1 -1873.115,E2 -1873.115} C_VEL
LIN {X 0,Y 580.525,Z 343.806,A -85,B 0,C 180,E1 -1876.167,E2 -1876.167} C_VEL
LIN {X 0,Y 580.555,Z 345.649,A -85,B 0,C 180,E1 -1876.324,E2 -1876.324} C_VEL
LIN {X 0,Y 580.978,Z 350.721,A -85,B 0,C 180,E1 -1876.401,E2 -1876.401} C_VEL
LIN {X 0,Y 580.805,Z 454.946,A -85,B 0,C 180,E1 -1877.708,E2 -1877.708} C_VEL
LIN {X 0,Y 580.757,Z 468.219,A -85,B 0,C 180,E1 -1878.017,E2 -1878.017} C_VEL
LIN {X 0,Y 580.659,Z 480.373,A -85,B 0,C 180,E1 -1878.436,E2 -1878.436} C_VEL
LIN {X 0,Y 580.564,Z 492.628,A -85,B 0,C 180,E1 -1879.009,E2 -1879.009} C_VEL
LIN {X 0,Y 580.444,Z 504.202,A -85,B 0,C 180,E1 -1879.712,E2 -1879.712} C_VEL
LIN {X 0,Y 580.343,Z 514.599,A -85,B 0,C 180,E1 -1880.503,E2 -1880.503} C_VEL
LIN {X 0,Y 580.271,Z 523.111,A -85,B 0,C 180,E1 -1881.292,E2 -1881.292} C_VEL
LIN {X 0,Y 580.222,Z 530.96,A -85,B 0,C 180,E1 -1882.168,E2 -1882.168} C_VEL
LIN {X 0,Y 580.154,Z 538.65,A -85,B 0,C 180,E1 -1883.221,E2 -1883.221} C_VEL
LIN {X 0,Y 580.139,Z 545.679,A -85,B 0,C 180,E1 -1884.438,E2 -1884.438} C_VEL
LIN {X 0,Y 580.108,Z 550.371,A -85,B 0,C 180,E1 -1885.483,E2 -1885.483} C_VEL
LIN {X 0,Y 580.123,Z 553.956,A -85,B 0,C 180,E1 -1886.527,E2 -1886.527} C_VEL
LIN {X 0,Y 580.043,Z 555.808,A -85,B 0,C 180,E1 -1887.222,E2 -1887.222} C_VEL
LIN {X 0,Y 580.04,Z 557.198,A -85,B 0,C 180,E1 -1887.917,E2 -1887.917} C_VEL
LIN {X 0,Y 580.04,Z 558.785,A -85,B 0,C 180,E1 -1889.305,E2 -1889.305} C_VEL
LIN {X 0,Y 580.037,Z 559,A -85,B 0,C 180,E1 -1890,E2 -1890} C_VEL
LIN {X 0,Y 580.047,Z 558.186,A -85,B 0,C 180,E1 -1891.388,E2 -1891.388} C_VEL
LIN {X 0,Y 580.04,Z 557.201,A -85,B 0,C 180,E1 -1892.083,E2 -1892.083} C_VEL
LIN {X 0,Y 580.043,Z 555.811,A -85,B 0,C 180,E1 -1892.778,E2 -1892.778} C_VEL
LIN {X 0,Y 580.109,Z 552.897,A -85,B 0,C 180,E1 -1893.82,E2 -1893.82} C_VEL
LIN {X 0,Y 580.054,Z 548.951,A -85,B 0,C 180,E1 -1894.865,E2 -1894.865} C_VEL
LIN {X 0,Y 580.139,Z 542.879,A -85,B 0,C 180,E1 -1896.084,E2 -1896.084} C_VEL
LIN {X 0,Y 580.184,Z 536.241,A -85,B 0,C 180,E1 -1897.132,E2 -1897.132} C_VEL
LIN {X 0,Y 580.25,Z 527.994,A -85,B 0,C 180,E1 -1898.181,E2 -1898.181} C_VEL
LIN {X 0,Y 580.307,Z 519.544,A -85,B 0,C 180,E1 -1899.058,E2 -1899.058} C_VEL
LIN {X 0,Y 580.425,Z 509.104,A -85,B 0,C 180,E1 -1899.935,E2 -1899.935} C_VEL
LIN {X 0,Y 580.494,Z 498.764,A -85,B 0,C 180,E1 -1900.639,E2 -1900.639} C_VEL
LIN {X 0,Y 580.597,Z 487.24,A -85,B 0,C 180,E1 -1901.264,E2 -1901.264} C_VEL
LIN {X 0,Y 580.676,Z 474.488,A -85,B 0,C 180,E1 -1901.784,E2 -1901.784} C_VEL
LIN {X 0,Y 580.774,Z 461.458,A -85,B 0,C 180,E1 -1902.159,E2 -1902.159} C_VEL
LIN {X 0,Y 580.831,Z 449.126,A -85,B 0,C 180,E1 -1902.379,E2 -1902.379} C_VEL
LIN {X 0,Y 580.844,Z 347.638,A -85,B 0,C 180,E1 -1903.641,E2 -1903.641} C_VEL
LIN {X 0,Y 580.514,Z 345.158,A -85,B 0,C 180,E1 -1903.699,E2 -1903.699} C_VEL
LIN {X 0,Y 580.695,Z 319.651,A -85,B 0,C 180,E1 -1906.523,E2 -1906.523} C_VEL
LIN {X 0,Y 580.933,Z 293.319,A -85,B 0,C 180,E1 -1909.495,E2 -1909.495} C_VEL
LIN {X 0,Y 581.215,Z 268.109,A -85,B 0,C 180,E1 -1912.388,E2 -1912.388} C_VEL
LIN {X 0,Y 581.344,Z 245.423,A -85,B 0,C 180,E1 -1914.947,E2 -1914.947} C_VEL
LIN {X 0,Y 581.234,Z 237.876,A -85,B 0,C 180,E1 -1915.803,E2 -1915.803} C_VEL
LIN {X 0,Y 580.275,Z 233.304,A -85,B 0,C 180,E1 -1916.391,E2 -1916.391} C_VEL
LIN {X 0,Y 580.24,Z 233.211,A -85,B 0,C 180,E1 -1919.298,E2 -1919.298} C_VEL
LIN {X 0,Y 580.27,Z 233.2,A -85,B 0,C 180,E1 -1922.201,E2 -1922.201} C_VEL
LIN {X 0,Y 580.262,Z 233.201,A -85,B 0,C 180,E1 -1924.697,E2 -1924.697} C_VEL
LIN {X 0,Y 580.257,Z 233.208,A -85,B 0,C 180,E1 -1927.27,E2 -1927.27} C_VEL
LIN {X 0,Y 580.26,Z 233.199,A -85,B 0,C 180,E1 -1930.267,E2 -1930.267} C_VEL
LIN {X 0,Y 580.236,Z 233.204,A -85,B 0,C 180,E1 -1932.709,E2 -1932.709} C_VEL
LIN {X 0,Y 580.237,Z 233.206,A -85,B 0,C 180,E1 -1935.611,E2 -1935.611} C_VEL
LIN {X 0,Y 580.225,Z 233.204,A -85,B 0,C 180,E1 -1938.226,E2 -1938.226} C_VEL
LIN {X 0,Y 580.249,Z 233.208,A -85,B 0,C 180,E1 -1940.963,E2 -1940.963} C_VEL
LIN {X 0,Y 580.225,Z 233.207,A -85,B 0,C 180,E1 -1943.593,E2 -1943.593} C_VEL
LIN {X 0,Y 580.254,Z 233.2,A -85,B 0,C 180,E1 -1946.141,E2 -1946.141} C_VEL
LIN {X 0,Y 580.238,Z 233.206,A -85,B 0,C 180,E1 -1948.612,E2 -1948.612} C_VEL
LIN {X 0,Y 580.25,Z 233.21,A -85,B 0,C 180,E1 -1951.022,E2 -1951.022} C_VEL
LIN {X 0,Y 580.24,Z 233.203,A -85,B 0,C 180,E1 -1953.673,E2 -1953.673} C_VEL
LIN {X 0,Y 580.229,Z 233.206,A -85,B 0,C 180,E1 -1956.44,E2 -1956.44} C_VEL
LIN {X 0,Y 580.237,Z 233.204,A -85,B 0,C 180,E1 -1959.436,E2 -1959.436} C_VEL
LIN {X 0,Y 580.22,Z 233.205,A -85,B 0,C 180,E1 -1961.644,E2 -1961.644} C_VEL
LIN {X 0,Y 580.228,Z 233.203,A -85,B 0,C 180,E1 -1963.824,E2 -1963.824} C_VEL
LIN {X 0,Y 580.266,Z 233.199,A -85,B 0,C 180,E1 -1965.982,E2 -1965.982} C_VEL
LIN {X 0,Y 580.291,Z 233.204,A -85,B 0,C 180,E1 -1968.827,E2 -1968.827} C_VEL
LIN {X 0,Y 580.268,Z 233.198,A -85,B 0,C 180,E1 -1971.643,E2 -1971.643} C_VEL
LIN {X 0,Y 580.294,Z 233.203,A -85,B 0,C 180,E1 -1974.44,E2 -1974.44} C_VEL
LIN {X 0,Y 580.295,Z 233.196,A -85,B 0,C 180,E1 -1977.223,E2 -1977.223} C_VEL
LIN {X 0,Y 580.312,Z 233.196,A -85,B 0,C 180,E1 -1980,E2 -1980} C_VEL
LIN {X 0,Y 580.312,Z 233.198,A -85,B 0,C 180,E1 -1982.777,E2 -1982.777} C_VEL
LIN {X 0,Y 580.272,Z 233.198,A -85,B 0,C 180,E1 -1985.56,E2 -1985.56} C_VEL
LIN {X 0,Y 580.275,Z 233.208,A -85,B 0,C 180,E1 -1988.357,E2 -1988.357} C_VEL
LIN {X 0,Y 580.252,Z 233.201,A -85,B 0,C 180,E1 -1991.174,E2 -1991.174} C_VEL
LIN {X 0,Y 580.282,Z 233.202,A -85,B 0,C 180,E1 -1994.018,E2 -1994.018} C_VEL
LIN {X 0,Y 580.253,Z 233.201,A -85,B 0,C 180,E1 -1996.899,E2 -1996.899} C_VEL
LIN {X 0,Y 580.259,Z 233.204,A -85,B 0,C 180,E1 -1999.824,E2 -1999.824} C_VEL
LIN {X 0,Y 580.259,Z 233.2,A -85,B 0,C 180,E1 -2001.33,E2 -2001.33} C_VEL
LIN {X 0,Y 579.556,Z 233.295,A -85,B 0,C 180,E1 -2001.909,E2 -2001.909} C_VEL
LIN {X 0,Y 576.681,Z 233.649,A -85,B 0,C 180,E1 -2002.849,E2 -2002.849} C_VEL
LIN {X 0,Y 574.284,Z 233.947,A -85,B 0,C 180,E1 -2003.605,E2 -2003.605} C_VEL
LIN {X 0,Y 573.273,Z 234.079,A -85,B 0,C 180,E1 -2004.189,E2 -2004.189} C_VEL
LIN {X 0,Y 573.2,Z 234.081,A -85,B 0,C 180,E1 -2004.386,E2 -2004.386} C_VEL
LIN {X 0,Y 573.169,Z 234.083,A -85,B 0,C 180,E1 -2006.98,E2 -2006.98} C_VEL
LIN {X 0,Y 573.213,Z 234.085,A -85,B 0,C 180,E1 -2010.178,E2 -2010.178} C_VEL
LIN {X 0,Y 573.211,Z 234.079,A -85,B 0,C 180,E1 -2012.648,E2 -2012.648} C_VEL
LIN {X 0,Y 573.172,Z 234.083,A -85,B 0,C 180,E1 -2015.191,E2 -2015.191} C_VEL
LIN {X 0,Y 573.201,Z 234.088,A -85,B 0,C 180,E1 -2017.811,E2 -2017.811} C_VEL
LIN {X 0,Y 573.192,Z 234.081,A -85,B 0,C 180,E1 -2020.53,E2 -2020.53} C_VEL
LIN {X 0,Y 573.18,Z 234.085,A -85,B 0,C 180,E1 -2023.365,E2 -2023.365} C_VEL
LIN {X 0,Y 573.197,Z 234.081,A -85,B 0,C 180,E1 -2026.337,E2 -2026.337} C_VEL
LIN {X 0,Y 573.18,Z 234.082,A -85,B 0,C 180,E1 -2028.54,E2 -2028.54} C_VEL
LIN {X 0,Y 573.22,Z 234.081,A -85,B 0,C 180,E1 -2031.298,E2 -2031.298} C_VEL
LIN {X 0,Y 573.177,Z 234.085,A -85,B 0,C 180,E1 -2034.024,E2 -2034.024} C_VEL
LIN {X 0,Y 573.219,Z 234.077,A -85,B 0,C 180,E1 -2036.516,E2 -2036.516} C_VEL
LIN {X 0,Y 573.192,Z 234.084,A -85,B 0,C 180,E1 -2039.125,E2 -2039.125} C_VEL
LIN {X 0,Y 573.191,Z 234.089,A -85,B 0,C 180,E1 -2041.434,E2 -2041.434} C_VEL
LIN {X 0,Y 573.218,Z 234.081,A -85,B 0,C 180,E1 -2043.809,E2 -2043.809} C_VEL
LIN {X 0,Y 573.213,Z 234.079,A -85,B 0,C 180,E1 -2046.862,E2 -2046.862} C_VEL
LIN {X 0,Y 573.229,Z 234.082,A -85,B 0,C 180,E1 -2049.174,E2 -2049.174} C_VEL
LIN {X 0,Y 573.19,Z 234.089,A -85,B 0,C 180,E1 -2051.411,E2 -2051.411} C_VEL
LIN {X 0,Y 573.215,Z 234.082,A -85,B 0,C 180,E1 -2053.621,E2 -2053.621} C_VEL
LIN {X 0,Y 573.192,Z 234.081,A -85,B 0,C 180,E1 -2056.529,E2 -2056.529} C_VEL
LIN {X 0,Y 573.236,Z 234.083,A -85,B 0,C 180,E1 -2059.403,E2 -2059.403} C_VEL
LIN {X 0,Y 573.202,Z 234.082,A -85,B 0,C 180,E1 -2062.249,E2 -2062.249} C_VEL
LIN {X 0,Y 573.251,Z 234.255,A -85,B 0,C 180,E1 -2064.328,E2 -2064.328} C_VEL
LIN {X 0,Y 573.508,Z 235.305,A -85,B 0,C 180,E1 -2064.441,E2 -2064.441} C_VEL
LIN {X 0,Y 574.077,Z 237.465,A -85,B 0,C 180,E1 -2064.49,E2 -2064.49} C_VEL
LIN {X 0,Y 573.867,Z 325.377,A -85,B 0,C 180,E1 -2065.611,E2 -2065.611} C_VEL
LIN {X 0,Y 573.798,Z 339.074,A -85,B 0,C 180,E1 -2065.94,E2 -2065.94} C_VEL
LIN {X 0,Y 573.694,Z 351.899,A -85,B 0,C 180,E1 -2066.401,E2 -2066.401} C_VEL
LIN {X 0,Y 573.538,Z 364.358,A -85,B 0,C 180,E1 -2067.015,E2 -2067.015} C_VEL
LIN {X 0,Y 573.417,Z 375.466,A -85,B 0,C 180,E1 -2067.717,E2 -2067.717} C_VEL
LIN {X 0,Y 573.315,Z 385.513,A -85,B 0,C 180,E1 -2068.508,E2 -2068.508} C_VEL
LIN {X 0,Y 573.225,Z 395.395,A -85,B 0,C 180,E1 -2069.473,E2 -2069.473} C_VEL
LIN {X 0,Y 573.133,Z 404.125,A -85,B 0,C 180,E1 -2070.527,E2 -2070.527} C_VEL
LIN {X 0,Y 573.065,Z 411.145,A -85,B 0,C 180,E1 -2071.581,E2 -2071.581} C_VEL
LIN {X 0,Y 572.986,Z 417.574,A -85,B 0,C 180,E1 -2072.812,E2 -2072.812} C_VEL
LIN {X 0,Y 573.015,Z 421.83,A -85,B 0,C 180,E1 -2073.868,E2 -2073.868} C_VEL
LIN {X 0,Y 572.943,Z 425.042,A -85,B 0,C 180,E1 -2074.926,E2 -2074.926} C_VEL
LIN {X 0,Y 573,Z 426.639,A -85,B 0,C 180,E1 -2075.631,E2 -2075.631} C_VEL
LIN {X 0,Y 573.013,Z 428.084,A -85,B 0,C 180,E1 -2076.55,E2 -2076.55} C_VEL
LIN {X 0,Y 572.978,Z 428.942,A -85,B 0,C 180,E1 -2077.754,E2 -2077.754} C_VEL
LIN {X 0,Y 572.951,Z 428.912,A -85,B 0,C 180,E1 -2078.465,E2 -2078.465} C_VEL
LIN {X 0,Y 572.926,Z 428.486,A -85,B 0,C 180,E1 -2079.176,E2 -2079.176} C_VEL
LIN {X 0,Y 572.975,Z 427.618,A -85,B 0,C 180,E1 -2079.888,E2 -2079.888} C_VEL
LIN {X 0,Y 572.988,Z 425.171,A -85,B 0,C 180,E1 -2081.112,E2 -2081.112} C_VEL
LIN {X 0,Y 573.012,Z 421.223,A -85,B 0,C 180,E1 -2082.394,E2 -2082.394} C_VEL
LIN {X 0,Y 573.033,Z 416.668,A -85,B 0,C 180,E1 -2083.475,E2 -2083.475} C_VEL
LIN {X 0,Y 573.095,Z 409.759,A -85,B 0,C 180,E1 -2084.732,E2 -2084.732} C_VEL
LIN {X 0,Y 573.129,Z 402.055,A -85,B 0,C 180,E1 -2085.833,E2 -2085.833} C_VEL
LIN {X 0,Y 573.189,Z 394.658,A -85,B 0,C 180,E1 -2086.697,E2 -2086.697} C_VEL
LIN {X 0,Y 573.381,Z 384.59,A -85,B 0,C 180,E1 -2087.66,E2 -2087.66} C_VEL
LIN {X 0,Y 573.449,Z 373.784,A -85,B 0,C 180,E1 -2088.488,E2 -2088.488} C_VEL
LIN {X 0,Y 573.572,Z 362.133,A -85,B 0,C 180,E1 -2089.199,E2 -2089.199} C_VEL
LIN {X 0,Y 573.675,Z 350.342,A -85,B 0,C 180,E1 -2089.753,E2 -2089.753} C_VEL
LIN {X 0,Y 573.804,Z 336.699,A -85,B 0,C 180,E1 -2090.22,E2 -2090.22} C_VEL
LIN {X 0,Y 573.904,Z 324.421,A -85,B 0,C 180,E1 -2090.497,E2 -2090.497} C_VEL
LIN {X 0,Y 574.036,Z 236.996,A -85,B 0,C 180,E1 -2091.607,E2 -2091.607} C_VEL
LIN {X 0,Y 573.366,Z 234.823,A -85,B 0,C 180,E1 -2091.681,E2 -2091.681} C_VEL
LIN {X 0,Y 573.234,Z 234.12,A -85,B 0,C 180,E1 -2091.817,E2 -2091.817} C_VEL
LIN {X 0,Y 573.226,Z 234.084,A -85,B 0,C 180,E1 -2094.636,E2 -2094.636} C_VEL
LIN {X 0,Y 573.19,Z 234.09,A -85,B 0,C 180,E1 -2096.979,E2 -2096.979} C_VEL
LIN {X 0,Y 573.222,Z 234.078,A -85,B 0,C 180,E1 -2099.483,E2 -2099.483} C_VEL
LIN {X 0,Y 573.25,Z 234.073,A -85,B 0,C 180,E1 -2102.227,E2 -2102.227} C_VEL
LIN {X 0,Y 573.225,Z 234.082,A -85,B 0,C 180,E1 -2104.769,E2 -2104.769} C_VEL
LIN {X 0,Y 573.216,Z 234.075,A -85,B 0,C 180,E1 -2107.808,E2 -2107.808} C_VEL
LIN {X 0,Y 573.245,Z 234.083,A -85,B 0,C 180,E1 -2110.524,E2 -2110.524} C_VEL
LIN {X 0,Y 573.205,Z 234.079,A -85,B 0,C 180,E1 -2113.361,E2 -2113.361} C_VEL
LIN {X 0,Y 573.202,Z 234.086,A -85,B 0,C 180,E1 -2116.335,E2 -2116.335} C_VEL
LIN {X 0,Y 573.242,Z 234.074,A -85,B 0,C 180,E1 -2119.474,E2 -2119.474} C_VEL
LIN {X 0,Y 573.215,Z 234.083,A -85,B 0,C 180,E1 -2122.19,E2 -2122.19} C_VEL
LIN {X 0,Y 573.218,Z 234.077,A -85,B 0,C 180,E1 -2125.23,E2 -2125.23} C_VEL
LIN {X 0,Y 573.24,Z 234.076,A -85,B 0,C 180,E1 -2127.772,E2 -2127.772} C_VEL
LIN {X 0,Y 573.252,Z 234.075,A -85,B 0,C 180,E1 -2130.633,E2 -2130.633} C_VEL
LIN {X 0,Y 573.194,Z 234.081,A -85,B 0,C 180,E1 -2133.514,E2 -2133.514} C_VEL
LIN {X 0,Y 573.219,Z 234.083,A -85,B 0,C 180,E1 -2136.134,E2 -2136.134} C_VEL
LIN {X 0,Y 573.238,Z 234.07,A -85,B 0,C 180,E1 -2139.173,E2 -2139.173} C_VEL
LIN {X 0,Y 573.197,Z 234.08,A -85,B 0,C 180,E1 -2141.41,E2 -2141.41} C_VEL
LIN {X 0,Y 573.219,Z 234.081,A -85,B 0,C 180,E1 -2143.621,E2 -2143.621} C_VEL
LIN {X 0,Y 573.247,Z 234.08,A -85,B 0,C 180,E1 -2145.806,E2 -2145.806} C_VEL
LIN {X 0,Y 573.255,Z 234.072,A -85,B 0,C 180,E1 -2148.745,E2 -2148.745} C_VEL
LIN {X 0,Y 573.237,Z 234.078,A -85,B 0,C 180,E1 -2151.54,E2 -2151.54} C_VEL
LIN {X 0,Y 573.255,Z 234.073,A -85,B 0,C 180,E1 -2154.371,E2 -2154.371} C_VEL
LIN {X 0,Y 573.287,Z 234.075,A -85,B 0,C 180,E1 -2157.892,E2 -2157.892} C_VEL
LIN {X 0,Y 573.297,Z 234.071,A -85,B 0,C 180,E1 -2160,E2 -2160} C_VEL
LIN {X 0,Y 573.272,Z 234.069,A -85,B 0,C 180,E1 -2162.811,E2 -2162.811} C_VEL
LIN {X 0,Y 573.266,Z 234.079,A -85,B 0,C 180,E1 -2165.628,E2 -2165.628} C_VEL
LIN {X 0,Y 573.224,Z 234.075,A -85,B 0,C 180,E1 -2168.46,E2 -2168.46} C_VEL
LIN {X 0,Y 573.263,Z 234.079,A -85,B 0,C 180,E1 -2171.312,E2 -2171.312} C_VEL
LIN {X 0,Y 573.234,Z 234.074,A -85,B 0,C 180,E1 -2174.409,E2 -2174.409} C_VEL
LIN {X 0,Y 573.237,Z 234.081,A -85,B 0,C 180,E1 -2177.112,E2 -2177.112} C_VEL
LIN {X 0,Y 573.22,Z 234.077,A -85,B 0,C 180,E1 -2180.078,E2 -2180.078} C_VEL
LIN {X 0,Y 573.207,Z 234.078,A -85,B 0,C 180,E1 -2182.339,E2 -2182.339} C_VEL
LIN {X 0,Y 573.212,Z 234.083,A -85,B 0,C 180,E1 -2185.412,E2 -2185.412} C_VEL
LIN {X 0,Y 573.191,Z 234.078,A -85,B 0,C 180,E1 -2188.019,E2 -2188.019} C_VEL
LIN {X 0,Y 573.209,Z 234.078,A -85,B 0,C 180,E1 -2190.178,E2 -2190.178} C_VEL
LIN {X 0,Y 573.236,Z 234.078,A -85,B 0,C 180,E1 -2192.646,E2 -2192.646} C_VEL
LIN {X 0,Y 573.18,Z 234.089,A -85,B 0,C 180,E1 -2195.19,E2 -2195.19} C_VEL
LIN {X 0,Y 573.209,Z 234.078,A -85,B 0,C 180,E1 -2197.81,E2 -2197.81} C_VEL
LIN {X 0,Y 573.24,Z 234.078,A -85,B 0,C 180,E1 -2200.526,E2 -2200.526} C_VEL
LIN {X 0,Y 573.197,Z 234.08,A -85,B 0,C 180,E1 -2203.665,E2 -2203.665} C_VEL
LIN {X 0,Y 573.188,Z 234.088,A -85,B 0,C 180,E1 -2206.637,E2 -2206.637} C_VEL
LIN {X 0,Y 573.207,Z 234.078,A -85,B 0,C 180,E1 -2209.48,E2 -2209.48} C_VEL
LIN {X 0,Y 573.185,Z 234.083,A -85,B 0,C 180,E1 -2212.189,E2 -2212.189} C_VEL
LIN {X 0,Y 573.21,Z 234.079,A -85,B 0,C 180,E1 -2215.233,E2 -2215.233} C_VEL
LIN {X 0,Y 573.219,Z 234.077,A -85,B 0,C 180,E1 -2217.777,E2 -2217.777} C_VEL
LIN {X 0,Y 573.21,Z 234.086,A -85,B 0,C 180,E1 -2220.631,E2 -2220.631} C_VEL
LIN {X 0,Y 573.216,Z 234.21,A -85,B 0,C 180,E1 -2223.495,E2 -2223.495} C_VEL
LIN {X 0,Y 574.38,Z 240.309,A -85,B 0,C 180,E1 -2224.255,E2 -2224.255} C_VEL
LIN {X 0,Y 574.311,Z 263.074,A -85,B 0,C 180,E1 -2226.825,E2 -2226.825} C_VEL
LIN {X 0,Y 574.17,Z 284.21,A -85,B 0,C 180,E1 -2229.209,E2 -2229.209} C_VEL
LIN {X 0,Y 573.866,Z 309.982,A -85,B 0,C 180,E1 -2232.172,E2 -2232.172} C_VEL
LIN {X 0,Y 573.598,Z 335.753,A -85,B 0,C 180,E1 -2235.09,E2 -2235.09} C_VEL
LIN {X 0,Y 573.513,Z 345.15,A -85,B 0,C 180,E1 -2236.13,E2 -2236.13} C_VEL
LIN {X 0,Y 574.078,Z 350.721,A -85,B 0,C 180,E1 -2236.234,E2 -2236.234} C_VEL
LIN {X 0,Y 573.881,Z 454.945,A -85,B 0,C 180,E1 -2237.557,E2 -2237.557} C_VEL
LIN {X 0,Y 573.8,Z 468.218,A -85,B 0,C 180,E1 -2237.87,E2 -2237.87} C_VEL
LIN {X 0,Y 573.702,Z 481.152,A -85,B 0,C 180,E1 -2238.325,E2 -2238.325} C_VEL
LIN {X 0,Y 573.576,Z 492.721,A -85,B 0,C 180,E1 -2238.878,E2 -2238.878} C_VEL
LIN {X 0,Y 573.435,Z 504.2,A -85,B 0,C 180,E1 -2239.585,E2 -2239.585} C_VEL
LIN {X 0,Y 573.33,Z 514.6,A -85,B 0,C 180,E1 -2240.385,E2 -2240.385} C_VEL
LIN {X 0,Y 573.241,Z 523.112,A -85,B 0,C 180,E1 -2241.185,E2 -2241.185} C_VEL
LIN {X 0,Y 573.161,Z 530.96,A -85,B 0,C 180,E1 -2242.071,E2 -2242.071} C_VEL
